TYPE "UDT_ConveyorStatistics"
TITLE = UDT_ConveyorStatistics
VERSION : 0.1
//User-defined structure of FB_Conveyor function block statistics.
   STRUCT
      EnergySave : "UDT_EventStatistic";   // Number of times that save energy mode occurs
      ConveyorUp : "UDT_EventStatistic";   // Conveyor up statistics
      ConveyorDown : "UDT_EventStatistic";   // Conveyor down statistics
      ConveyorStop : "UDT_EventStatistic";   // Conveyor down statistics
   END_STRUCT;

END_TYPE

TYPE "UDT_ConveyorStatus"
TITLE = UDT_ConveyorStatus
VERSION : 0.1
//User-defined structure of FB_Conveyor function block status.
   STRUCT
      Status : Int;   // Status number
      Specific : Struct
         Reverse { ExternalAccessible := 'False'; ExternalVisible := 'False'; ExternalWritable := 'False'} : Bool;   // Conveyor is running in reverse direction
      END_STRUCT;
   END_STRUCT;

END_TYPE

TYPE "UDT_EncoderStatisticsV2"
VERSION : 0.1
   STRUCT
      RunningFeedbackError : "UDT_EventStatistic";
      InvalidValue : "UDT_EventStatistic";
   END_STRUCT;

END_TYPE

TYPE "UDT_EncoderStatusV2"
VERSION : 0.1
   STRUCT
      InvalidValue : Bool;   // Invalid value
      RunningFeedbackError : Bool;   // Running feedback error
   END_STRUCT;

END_TYPE

TYPE "UDT_EncoderConfigurationV2"
VERSION : 0.1
   STRUCT
      EncoderMaxValue : DInt;   // The maximum value of the encoder where will rollover
      mmPerIncrement : Real;   // The mm per encoder incremental [mm]
      ErrorFilter : UDInt;   // Movment timeout without encoder data [ms]
      SamplingTime : UDInt;   // Save actual speed sampling time [ms]
   END_STRUCT;

END_TYPE

TYPE "UDT_EuchnerLockStatusV2"
VERSION : 0.1
   STRUCT
      LockFault : Bool;   // Internal lock fault
      DoorClosed : Bool;   // The door is closed
      DoorOpened : Bool;   // The door is opened
      BoltTongueClosed : Bool;   // The lock bolt tongue is closed
      ReqMissingAccessRights : Bool;   // Button access request triggered without permission from DHL
      ResetMissingAccessRights : Bool;   // Button reset triggered without permission from DHL
      DoorOpenedWithoutReq : Bool;   // Doors were opened without request and permission
      Safelylocked : Bool;   // The lock is safely locked
      SafetyLockAckReq : Bool;   // The safety lock signal needs to be confirmed
   END_STRUCT;

END_TYPE

TYPE "UDT_ConveyorCommand"
TITLE = UDT_ConveyorCommand
VERSION : 0.1
//User-defined structure of conveyor commands.
   STRUCT
      ManualMode { ExternalAccessible := 'False'; ExternalVisible := 'False'; ExternalWritable := 'False'} : Bool;   // Manual mode command from HMI
      ManualStartStop { ExternalAccessible := 'False'; ExternalVisible := 'False'; ExternalWritable := 'False'} : Bool;   // Run conveyor in manual mode
      ManualFullSpeed { ExternalAccessible := 'False'; ExternalVisible := 'False'; ExternalWritable := 'False'} : Bool;   // Full speed conveyor in manual mode
      ManualJog { ExternalAccessible := 'False'; ExternalVisible := 'False'; ExternalWritable := 'False'} : Bool;   // Command to jog conveyor in slow speed from HMI
      Reverse { ExternalAccessible := 'False'; ExternalVisible := 'False'; ExternalWritable := 'False'} : Bool;   // Command to run conveyor in reverse direction from HMI
      ManualSpeed : Int := 50;   // Manual mode speed as percentage of nominal speed [0-100%]
   END_STRUCT;

END_TYPE

TYPE "UDT_Outfeed2StatesConfiguration"
VERSION : 0.1
//User-defined structure of FB_Chute2PEC function block configuration.
   STRUCT
      FullDetectionTime : UDInt;   // Time after which chute full is detected
      FullReleaseTime : UDInt;   // Time after which chute full is released
      HalfFullDetectionTime : UDInt;   // Time after which chute half full is detected
      HalfFullReleaseTime : UDInt;   // Time after which chute half full is released
   END_STRUCT;

END_TYPE

TYPE "UDT_ConveyorConfiguration"
TITLE = UDT_ConveyorConfiguration
VERSION : 0.1
//User-defined structure of conveyor parameters.
   STRUCT
      Common : "UDT_ConveyorCommonConfiguration";   // Common configuration
      Forward_Direction : Struct   // Forward Direction configuration
         EnergySaveLenght : DInt;   // Distance conveyor travelled before energy save activate [cm]
         GapHeadToHead : DInt;   // Gapping head to head value [cm]
         GapTailToHead : DInt;   // Gapping tail to head value [cm]
         GapCorrection : DInt;   // Gap offset to cover VFD's ramps [cm]
         PEC_EoSDistanceOffset : DInt;   // Distance offset between photo eye and the end of conveyor [mm]
         Mode : Int;   // Automatic operation; 1- Slave; 2- Queue;
         FirstConveyorToStart { ExternalAccessible := 'False'; ExternalVisible := 'False'; ExternalWritable := 'False'} : Bool;   // First conveyor to start cascade mode forward direction
      END_STRUCT;
      Reverse_Direction : Struct   // Reverse Direction configuration
         EnergySaveLenght : DInt;   // Distance conveyor travelled before energy save activate [cm]
         GapHeadToHead : DInt;   // Gapping head to head value [cm]
         GapTailToHead : DInt;   // Gapping tail to head value [cm]
         GapCorrection : DInt;   // Gap offset to cover VFD's ramps [cm]
         PEC_BoSDistanceOffset : DInt;   // Distance offset between photo eye and the end of conveyor [mm]
         Mode : Int;   // Automatic operation; 1- Slave; 2- Queue;
         FirstConveyorToStart { ExternalAccessible := 'False'; ExternalVisible := 'False'; ExternalWritable := 'False'} : Bool;   // First conveyor to start cascade mode reverse direction
      END_STRUCT;
      CascadeTimeOnDelay : UDInt;   // Cascade time on delay [ms]
      ExtraGapRecovery : DInt;   // Extra gap to recovery die back [cm]
      SpeedSetpointLow : Int;   // Low speed setpoint [mm/s]
      SpeedSetpointNominal : Int;   // Nominal speed setpoint [mm/s]
      Energy { ExternalAccessible := 'False'; ExternalVisible := 'False'; ExternalWritable := 'False'} : Bool;   // Energy save mode enable
      Bi_Directional_Enable { ExternalAccessible := 'False'; ExternalVisible := 'False'; ExternalWritable := 'False'} : Bool;   // The conveyor can run in both directions
   END_STRUCT;

END_TYPE

TYPE "UDT_SerialCommunicationStatus"
VERSION : 0.1
   STRUCT
      ErrorCode : Word;   // Siemens Signal_Get error code - Check documetation
      Connected : Bool;   // Connected
      CommunicationFault : Bool;   // Communication fault
   END_STRUCT;

END_TYPE

TYPE "UDT_XrayInterface"
VERSION : 0.1
   STRUCT
      Backbelt : Struct   // Bacbelt function signals structure
         Enable : Bool;   // TRUE when Backbelt functionality for input conveyor is active
         Active : Bool;   // TRUE when Backbelt functionality activeted
      END_STRUCT;
      XrayConveyor : Struct   // Xray conveyor signals structure
         RunFwd : Bool;   // TRUE when conveyor is running forward
         RunRvs : Bool;   // TRUE when conveyor is running reverse
      END_STRUCT;
      InputConveyor : Struct   // Input conveyor signals structure
         CommandRunRvs : Bool;   // Request command to run reverse
      END_STRUCT;
      Communication : Struct   // SerialCommunication signals structure
         Connceted : Bool;   // Devices connected
         SendMessage : Struct   // Send message signal structure
            SendTrigger : Bool;   // Send message trigger
            GIN : Int;   // GIN number for new message
         END_STRUCT;
      END_STRUCT;
   END_STRUCT;

END_TYPE

FUNCTION_BLOCK "FB_VFD_MultiControl_V4"
{ S7_Optimized_Access := 'TRUE' }
AUTHOR : 'KBA-PM'
VERSION : 0.1
// ATTRIBUTES
// AUTO_NUMBER = True
// BLOCK_NUMBER = 107
// END_ATTRIBUTES
   VAR_INPUT
      i_UDT_VFDConfiguration { ExternalAccessible := 'False'; ExternalVisible := 'False'; ExternalWritable := 'False'} : "UDT_VFD_MultiControl_Configuration";   //   VFD configuration structure
      i_UDT_VFDInputs { ExternalAccessible := 'False'; ExternalVisible := 'False'; ExternalWritable := 'False'} : "UDT_VFD_MultiControl_PI";   //   VFD inputs structure
      ix_PowerOK { ExternalAccessible := 'False'; ExternalVisible := 'False'; ExternalWritable := 'False'} : Bool;   //   TRUE when External Power OK
      ix_SafetyOK { ExternalAccessible := 'False'; ExternalVisible := 'False'; ExternalWritable := 'False'} : Bool;   //   TRUE when Safety OK
      ix_SimulationModeActive { ExternalAccessible := 'False'; ExternalVisible := 'False'; ExternalWritable := 'False'} : Bool;   //   TRUE when Simulation mode active
   END_VAR

   VAR_OUTPUT
      q_UDT_HMIStatus { ExternalAccessible := 'False'; ExternalVisible := 'False'; ExternalWritable := 'False'} : "UDT_VfdStatus";   //   HMI status structure
      qsi_UDT_VFDSpeed { ExternalAccessible := 'False'; ExternalVisible := 'False'; ExternalWritable := 'False'} : SInt;   //   VFD speed setpoint
   END_VAR

   VAR_IN_OUT
      iq_UDT_ConveyorInterface : "UDT_ConveyorInterface";   //   Conveyor interface structure
      iq_UDT_VFDStatistics : "UDT_VfdStatistics";   //   Statistics structure
      iq_UDT_Equipment : "UDT_EquipmentControl";   //   Equipment structure
   END_VAR

   VAR
      s_FB_TimerOnOffDelayCheckSupply { ExternalAccessible := 'False'; ExternalVisible := 'False'; ExternalWritable := 'False'; S7_SetPoint := 'False'} : "FB_TimerOnOffDelay";   //  "TimerOnOffDelay" - to delay time for VFD supply contactor
      s_FB_TimerOnOffDelay_ProfinetNotOnlineMasking { ExternalAccessible := 'False'; ExternalVisible := 'False'; ExternalWritable := 'False'; S7_SetPoint := 'False'} : "FB_TimerOnOffDelay";   //   "TimerOnOffDelay" - to delay time for profinet not online masking
      s_FB_TimerOnOffDelay_ProfinetSlaveErrorMasking { ExternalAccessible := 'False'; ExternalVisible := 'False'; ExternalWritable := 'False'; S7_SetPoint := 'False'} : "FB_TimerOnOffDelay";   //   "TimerOnOffDelay" - to delay time for profinet error masking
      s_FB_TimerOnOffDelay_RunCommand_Motor_1 { ExternalAccessible := 'False'; ExternalVisible := 'False'; ExternalWritable := 'False'; S7_SetPoint := 'False'} : "FB_TimerOnOffDelay";   //   "TimerOnOffDelay" - to delay time for run command motor 1
      s_FB_TimerOnOffDelay_RunCommand_Motor_2 { ExternalAccessible := 'False'; ExternalVisible := 'False'; ExternalWritable := 'False'; S7_SetPoint := 'False'} : "FB_TimerOnOffDelay";   //   "TimerOnOffDelay" - to delay time for run command motor 2
      s_FB_TimerOnOffDelay_RunCommand_Motor_3 { ExternalAccessible := 'False'; ExternalVisible := 'False'; ExternalWritable := 'False'; S7_SetPoint := 'False'} : "FB_TimerOnOffDelay";   //   "TimerOnOffDelay" - to delay time for run command motor 3
      s_FB_TimerOnOffDelay_SafetyOK { ExternalAccessible := 'False'; ExternalVisible := 'False'; ExternalWritable := 'False'; S7_SetPoint := 'False'} : "FB_TimerOnOffDelay";   //   "TimerOnOffDelay" - to delay time for safety
      s_FB_TimerOnOffDelay_RunCommand_Motor_4 { ExternalAccessible := 'False'; ExternalVisible := 'False'; ExternalWritable := 'False'; S7_SetPoint := 'False'} : "FB_TimerOnOffDelay";   //   "TimerOnOffDelay" - to delay time for run command motor 4
      s_FB_TimerOnOffDelay_Instance { ExternalAccessible := 'False'; ExternalVisible := 'False'; ExternalWritable := 'False'; S7_SetPoint := 'False'} : "FB_TimerOnOffDelay";   //   "TimerOnOffDelay" - to delay time for Instance
      s_UDT_HMIStatus { ExternalAccessible := 'False'; ExternalVisible := 'False'; ExternalWritable := 'False'; S7_SetPoint := 'False'} : "UDT_VfdStatus";   //   HMI status structure
      s_UDT_PNDevice { ExternalAccessible := 'False'; ExternalVisible := 'False'; ExternalWritable := 'False'; S7_SetPoint := 'False'} : "UDT_PNDevice";   //   PN device info structure
      s_R_TRIG_RunForward {InstructionName := 'R_TRIG'; LibVersion := '1.0'; ExternalAccessible := 'False'; ExternalVisible := 'False'; ExternalWritable := 'False'; S7_SetPoint := 'False'} : R_TRIG;   //   Rising edge of Run forward signal
      s_R_TRIG_RunReverse {InstructionName := 'R_TRIG'; LibVersion := '1.0'; ExternalAccessible := 'False'; ExternalVisible := 'False'; ExternalWritable := 'False'; S7_SetPoint := 'False'} : R_TRIG;   //   Rising edge of Run reverse
      s_R_TRIG_PNSlaveNotOnline {InstructionName := 'R_TRIG'; LibVersion := '1.0'; ExternalAccessible := 'False'; ExternalVisible := 'False'; ExternalWritable := 'False'; S7_SetPoint := 'False'} : R_TRIG;   //   Rising edge for trigger Profinet slave not online statistics
      s_R_TRIG_PNSlaveError {InstructionName := 'R_TRIG'; LibVersion := '1.0'; ExternalAccessible := 'False'; ExternalVisible := 'False'; ExternalWritable := 'False'; S7_SetPoint := 'False'} : R_TRIG;   //   Rising edge for trigger Profinet slave error statistics
      s_R_TRIG_InternalError {InstructionName := 'R_TRIG'; LibVersion := '1.0'; ExternalAccessible := 'False'; ExternalVisible := 'False'; ExternalWritable := 'False'; S7_SetPoint := 'False'} : R_TRIG;   //   Rising edge for trigger Internal VFD Error statistics
      s_R_TRIG_Running {InstructionName := 'R_TRIG'; LibVersion := '1.0'; ExternalAccessible := 'False'; ExternalVisible := 'False'; ExternalWritable := 'False'; S7_SetPoint := 'False'} : R_TRIG;   //   Rising edge for starting of the running signal
      s_R_TRIG_Instance {InstructionName := 'R_TRIG'; LibVersion := '1.0'; ExternalAccessible := 'False'; ExternalVisible := 'False'; ExternalWritable := 'False'; S7_SetPoint := 'False'} : R_TRIG;   //   Raising edge for Instance
      s_R_TRIG_NewPNSlaveError {InstructionName := 'R_TRIG'; LibVersion := '1.0'; ExternalAccessible := 'False'; ExternalVisible := 'False'; ExternalWritable := 'False'; S7_SetPoint := 'False'} : R_TRIG;   //   New profinet slave error trigger
      s_R_TRIG_NewPNSlaveNotOnline {InstructionName := 'R_TRIG'; LibVersion := '1.0'; ExternalAccessible := 'False'; ExternalVisible := 'False'; ExternalWritable := 'False'; S7_SetPoint := 'False'} : R_TRIG;   //   New profinet slave not online trigger
      ss_RDREC { ExternalAccessible := 'False'; ExternalVisible := 'False'; ExternalWritable := 'False'} : Struct   //   Read error code record structure
         Valid { ExternalAccessible := 'False'; ExternalVisible := 'False'; ExternalWritable := 'False'} : Bool;   //      Read operation is done
         Busy { ExternalAccessible := 'False'; ExternalVisible := 'False'; ExternalWritable := 'False'} : Bool;   //      Read operation is in progress
         Error { ExternalAccessible := 'False'; ExternalVisible := 'False'; ExternalWritable := 'False'} : Bool;   //      Read operation has an error
         Status { ExternalAccessible := 'False'; ExternalVisible := 'False'; ExternalWritable := 'False'} : DWord;   //      Read operation status
         Lenght { ExternalAccessible := 'False'; ExternalVisible := 'False'; ExternalWritable := 'False'} : UInt;   //      Lenght of the read record
      END_STRUCT;
      ss_WRREC { ExternalAccessible := 'False'; ExternalVisible := 'False'; ExternalWritable := 'False'} : Struct   //   Write record structure
         Acceleration { ExternalAccessible := 'False'; ExternalVisible := 'False'; ExternalWritable := 'False'} : Struct   //      Acceleration
            REQ { ExternalAccessible := 'False'; ExternalVisible := 'False'; ExternalWritable := 'False'} : Bool;   //      Requirement
            Index { ExternalAccessible := 'False'; ExternalVisible := 'False'; ExternalWritable := 'False'} : DInt;   //      Index
            Done { ExternalAccessible := 'False'; ExternalVisible := 'False'; ExternalWritable := 'False'} : Bool;   //      Operation is done
            Busy { ExternalAccessible := 'False'; ExternalVisible := 'False'; ExternalWritable := 'False'} : Bool;   //      Write operation is in progress
            Error { ExternalAccessible := 'False'; ExternalVisible := 'False'; ExternalWritable := 'False'} : Bool;   //      Write operation has an error
            Status { ExternalAccessible := 'False'; ExternalVisible := 'False'; ExternalWritable := 'False'} : DWord;   //      Write operation status
            Data { ExternalAccessible := 'False'; ExternalVisible := 'False'; ExternalWritable := 'False'} : Word;   //      Data to write
         END_STRUCT;
         Deceleration { ExternalAccessible := 'False'; ExternalVisible := 'False'; ExternalWritable := 'False'} : Struct   //      Deceleration
            REQ { ExternalAccessible := 'False'; ExternalVisible := 'False'; ExternalWritable := 'False'} : Bool;   //      Requirement
            Index { ExternalAccessible := 'False'; ExternalVisible := 'False'; ExternalWritable := 'False'} : DInt;   //      Index
            Done { ExternalAccessible := 'False'; ExternalVisible := 'False'; ExternalWritable := 'False'} : Bool;   //      Operation is done
            Busy { ExternalAccessible := 'False'; ExternalVisible := 'False'; ExternalWritable := 'False'} : Bool;   //      Write operation is in progress
            Error { ExternalAccessible := 'False'; ExternalVisible := 'False'; ExternalWritable := 'False'} : Bool;   //      Write operation has an error
            Status { ExternalAccessible := 'False'; ExternalVisible := 'False'; ExternalWritable := 'False'} : DWord;   //      Write operation status
            Data { ExternalAccessible := 'False'; ExternalVisible := 'False'; ExternalWritable := 'False'} : Word;   //      Data to write
         END_STRUCT;
      END_STRUCT;
      ss_AccelerationDone { ExternalAccessible := 'False'; ExternalVisible := 'False'; ExternalWritable := 'False'} : Struct   //   Acceleration is written
         Motor_1 { ExternalAccessible := 'False'; ExternalVisible := 'False'; ExternalWritable := 'False'} : Bool;
         Motor_2 { ExternalAccessible := 'False'; ExternalVisible := 'False'; ExternalWritable := 'False'} : Bool;
         Motor_3 { ExternalAccessible := 'False'; ExternalVisible := 'False'; ExternalWritable := 'False'} : Bool;
         Motor_4 { ExternalAccessible := 'False'; ExternalVisible := 'False'; ExternalWritable := 'False'} : Bool;
         All { ExternalAccessible := 'False'; ExternalVisible := 'False'; ExternalWritable := 'False'} : Bool;
      END_STRUCT;
      ss_DecelerationDone { ExternalAccessible := 'False'; ExternalVisible := 'False'; ExternalWritable := 'False'} : Struct   //   Deceleration is written
         Motor_1 { ExternalAccessible := 'False'; ExternalVisible := 'False'; ExternalWritable := 'False'} : Bool;
         Motor_2 { ExternalAccessible := 'False'; ExternalVisible := 'False'; ExternalWritable := 'False'} : Bool;
         Motor_3 { ExternalAccessible := 'False'; ExternalVisible := 'False'; ExternalWritable := 'False'} : Bool;
         Motor_4 { ExternalAccessible := 'False'; ExternalVisible := 'False'; ExternalWritable := 'False'} : Bool;
         All { ExternalAccessible := 'False'; ExternalVisible := 'False'; ExternalWritable := 'False'} : Bool;
      END_STRUCT;
      s_VFDGeoStruct {InstructionName := 'GEOADDR'; LibVersion := '1.0'; ExternalAccessible := 'False'; ExternalVisible := 'False'; ExternalWritable := 'False'; S7_SetPoint := 'False'} : GEOADDR;   //   Geo structure indicate to telegram
      s_RDREC_ErrorCode {InstructionName := 'RDREC'; LibVersion := '1.0'; ExternalAccessible := 'False'; ExternalVisible := 'False'; ExternalWritable := 'False'; S7_SetPoint := 'False'} : RDREC;   //   Read error code record instruction
      s_WRREC_ACC {InstructionName := 'WRREC'; LibVersion := '1.1'; ExternalAccessible := 'False'; ExternalVisible := 'False'; ExternalWritable := 'False'; S7_SetPoint := 'False'} : WRREC;   //   Write acceleration record inctruction
      s_WRREC_DEC {InstructionName := 'WRREC'; LibVersion := '1.1'; ExternalAccessible := 'False'; ExternalVisible := 'False'; ExternalWritable := 'False'; S7_SetPoint := 'False'} : WRREC;   //   Write deceleration record instruction
      shw_VFD_Telegram { ExternalAccessible := 'False'; ExternalVisible := 'False'; ExternalWritable := 'False'} : HW_ANY;   //   Free telegram's HW_ID
      sr_MaximumSpeed { ExternalAccessible := 'False'; ExternalVisible := 'False'; ExternalWritable := 'False'} : Real;   //   Maximum speed [mm/s]
      sr_SpeedsetpointCorrected { ExternalAccessible := 'False'; ExternalVisible := 'False'; ExternalWritable := 'False'} : Real;   //   Speedsetpoint corrected with factor
      sw_ErrorCode { ExternalAccessible := 'False'; ExternalVisible := 'False'; ExternalWritable := 'False'} : Word;   //   VFD error code
      si_RequiredSpeedSetpoint { ExternalAccessible := 'False'; ExternalVisible := 'False'; ExternalWritable := 'False'} : Int;   //   Required speed setpoint
      si_ActualSpeed { ExternalAccessible := 'False'; ExternalVisible := 'False'; ExternalWritable := 'False'} : Int;   //   Actual speed in [mm/s]
      si_Log2GeoReturn { ExternalAccessible := 'False'; ExternalVisible := 'False'; ExternalWritable := 'False'} : Int;   //   Log2Geo function return
      si_Geo2LogReturn { ExternalAccessible := 'False'; ExternalVisible := 'False'; ExternalWritable := 'False'} : Int;   //   Geo2Log function return
      si_AccelerationSetpoint { ExternalAccessible := 'False'; ExternalVisible := 'False'; ExternalWritable := 'False'} : Int;   //   Acceleration setpoint value
      si_DecelerationSetpoint { ExternalAccessible := 'False'; ExternalVisible := 'False'; ExternalWritable := 'False'} : Int;   //   Deceleration setpoint value
      si_AccelerationOld { ExternalAccessible := 'False'; ExternalVisible := 'False'; ExternalWritable := 'False'} : Int;   //   Old acceleration value
      si_DecelerationOld { ExternalAccessible := 'False'; ExternalVisible := 'False'; ExternalWritable := 'False'} : Int;   //   Old deceleration value
      si_MotorNumber_Acc { ExternalAccessible := 'False'; ExternalVisible := 'False'; ExternalWritable := 'False'} : Int;   //   Motor number that is connected to the Multicontrol module [1,2,3 or 4]
      si_MotorNumber_Dec { ExternalAccessible := 'False'; ExternalVisible := 'False'; ExternalWritable := 'False'} : Int;   //   Motor number that is connected to the Multicontrol module [1,2,3 or 4]
      si_PNSlaveErrorCount { ExternalAccessible := 'False'; ExternalVisible := 'False'; ExternalWritable := 'False'} : Int;   //   Profinet slave error counter
      si_PNSlaveNotOnlineCount { ExternalAccessible := 'False'; ExternalVisible := 'False'; ExternalWritable := 'False'} : Int;   //   Profinet slave not online counter
      ssi_MotorSpeed { ExternalAccessible := 'False'; ExternalVisible := 'False'; ExternalWritable := 'False'} : SInt;   //   Motor speed value
      sx_ConfigurationError { ExternalAccessible := 'False'; ExternalVisible := 'False'; ExternalWritable := 'False'} : Bool;   //   Commissioning: configuration error
      sx_PNDeviceHealthy { ExternalAccessible := 'False'; ExternalVisible := 'False'; ExternalWritable := 'False'} : Bool;   //   Profinet device is online and error free
      sx_PowerOk { ExternalAccessible := 'False'; ExternalVisible := 'False'; ExternalWritable := 'False'} : Bool;   //   Communication, safety and power are available
      sx_VFD_Available { ExternalAccessible := 'False'; ExternalVisible := 'False'; ExternalWritable := 'False'} : Bool;   //   Hardware of VFD is ok
      sx_ErrorActive { ExternalAccessible := 'False'; ExternalVisible := 'False'; ExternalWritable := 'False'} : Bool;   //   Block has an error
      sx_MotorError { ExternalAccessible := 'False'; ExternalVisible := 'False'; ExternalWritable := 'False'} : Bool;   //   Motor error all
      sx_Motor_1_Error { ExternalAccessible := 'False'; ExternalVisible := 'False'; ExternalWritable := 'False'} : Bool;   //   Motor error 1
      sx_Motor_2_Error { ExternalAccessible := 'False'; ExternalVisible := 'False'; ExternalWritable := 'False'} : Bool;   //   Motor error 2
      sx_Motor_3_Error { ExternalAccessible := 'False'; ExternalVisible := 'False'; ExternalWritable := 'False'} : Bool;   //   Motor error 3
      sx_Motor_4_Error { ExternalAccessible := 'False'; ExternalVisible := 'False'; ExternalWritable := 'False'} : Bool;   //   Motor error 4
      sx_EnableOperation { ExternalAccessible := 'False'; ExternalVisible := 'False'; ExternalWritable := 'False'} : Bool;   //   Enable operation signal
      sx_RunVFDForward { ExternalAccessible := 'False'; ExternalVisible := 'False'; ExternalWritable := 'False'} : Bool;   //   Start VFD forward
      sx_RunVFDReverse { ExternalAccessible := 'False'; ExternalVisible := 'False'; ExternalWritable := 'False'} : Bool;   //   Start VFD backward
      sx_SpeedSetpointReached { ExternalAccessible := 'False'; ExternalVisible := 'False'; ExternalWritable := 'False'} : Bool;   //   Motor is running at requested speed
      sx_ErrorDone { ExternalAccessible := 'False'; ExternalVisible := 'False'; ExternalWritable := 'False'} : Bool;   //   Error code is read
      sx_SafetyOK { ExternalAccessible := 'False'; ExternalVisible := 'False'; ExternalWritable := 'False'} : Bool;   //   Safety ok
      sx_MaskingReset { ExternalAccessible := 'False'; ExternalVisible := 'False'; ExternalWritable := 'False'} : Bool;   //   Masking reset
      sx_PNSlaveError { ExternalAccessible := 'False'; ExternalVisible := 'False'; ExternalWritable := 'False'} : Bool;   //   Profinet slave error
      sx_PNSlaveNotOnline { ExternalAccessible := 'False'; ExternalVisible := 'False'; ExternalWritable := 'False'} : Bool;   //   Profinet slave not online
   END_VAR

   VAR CONSTANT
      ci_VFDArea : UInt := 1;   //   Area ID of IO Profinet devices
      ci_SubmoduleHWType : UInt := 5;   //   Submodule HW_type number
      ci_TelegramSlot : UInt := 2;   //   Free Siemens telegram slot
      ci_TelegramSubslot : UInt := 1;   //   Free Siemens telegram subslot
      cdi_ErrorCodeIndex : DInt := 17154;   //   Error code index
      cdi_AccelerationIndex : DInt := 18200;   //   Acceleration index
      cdi_DecelerationIndex : DInt := 18204;   //   Deceleration index
   END_VAR


BEGIN
	(*
	----------------------------------------------------------------------------------------
	|                                                                                      |
	|  Copyright  2023             FORTNA Europe BV                                        |
	|  All Rights Reserved         Netherlands                                             |
	|                                                                                      |
	----------------------------------------------------------------------------------------

	Version history:
	Date        | Version   | Author        | Remark
	----------------------------------------------------------------------------------------
	24/05/2023  | 1.0       | S.Nikodem     | Initial version for 4 motors | DHL Munich 2023
	13/03/2024  | 1.1       | S. Nieswiec   | Added to new baseline
	*)

	REGION 1 - Get Device Profinet number

	    // Getting information about Profinet Device.
	    "FC_GetDevicePN"(is_PNDeviceName := #i_UDT_VFDConfiguration.VFDPNDeviceName,
	                     ix_SimulationModeActive := #ix_SimulationModeActive,
	                     iqUDT_PND := #s_UDT_PNDevice);

	END_REGION

	REGION 2 - Motor validation

	    //Motor number 1
	    // Delay
	    #s_FB_TimerOnOffDelay_RunCommand_Motor_1(iudi_OnDelayTime := 1500,
	                                             ix_SignalToDelay :=
	                                             (#sx_RunVFDForward
	                                             OR #sx_RunVFDReverse)
	                                             AND #i_UDT_VFDInputs.CurrentMotor1 < #i_UDT_VFDConfiguration.MinimumCurrentWhenRunninng);

	    #ssi_MotorSpeed := #i_UDT_VFDInputs.SpeedMotor1;

	    IF (#s_FB_TimerOnOffDelay_RunCommand_Motor_1.qx_DelayedSignal AND #sx_EnableOperation) OR #i_UDT_VFDInputs.ErrorMotor1
	    THEN

	        #sx_Motor_1_Error := TRUE;

	    END_IF;

	    //Motor number 2
	    #s_FB_TimerOnOffDelay_RunCommand_Motor_2(iudi_OnDelayTime := 1500,
	                                             ix_SignalToDelay :=
	                                             (#sx_RunVFDForward
	                                             OR #sx_RunVFDReverse)
	                                             AND #i_UDT_VFDInputs.CurrentMotor2 < #i_UDT_VFDConfiguration.MinimumCurrentWhenRunninng);

	    #ssi_MotorSpeed := #i_UDT_VFDInputs.SpeedMotor2;

	    IF (#s_FB_TimerOnOffDelay_RunCommand_Motor_2.qx_DelayedSignal AND #sx_EnableOperation) OR #i_UDT_VFDInputs.ErrorMotor2

	    THEN

	        #sx_Motor_2_Error := TRUE;

	    END_IF;

	    //Motor number 3
	    #s_FB_TimerOnOffDelay_RunCommand_Motor_3(iudi_OnDelayTime := 1500,
	                                             ix_SignalToDelay :=
	                                             (#sx_RunVFDForward
	                                             OR #sx_RunVFDReverse)
	                                             AND #i_UDT_VFDInputs.CurrentMotor3 < #i_UDT_VFDConfiguration.MinimumCurrentWhenRunninng);

	    #ssi_MotorSpeed := #i_UDT_VFDInputs.SpeedMotor3;

	    IF (#s_FB_TimerOnOffDelay_RunCommand_Motor_3.qx_DelayedSignal AND #sx_EnableOperation) OR #i_UDT_VFDInputs.ErrorMotor3
	    THEN

	        #sx_Motor_3_Error := TRUE;

	    END_IF;

	    //Motor number 4
	    #s_FB_TimerOnOffDelay_RunCommand_Motor_4(iudi_OnDelayTime := 1500,
	                                             ix_SignalToDelay :=
	                                             (#sx_RunVFDForward
	                                             OR #sx_RunVFDReverse)
	                                             AND #i_UDT_VFDInputs.CurrentMotor4 < #i_UDT_VFDConfiguration.MinimumCurrentWhenRunninng);

	    #ssi_MotorSpeed := #i_UDT_VFDInputs.SpeedMotor4;

	    IF (#s_FB_TimerOnOffDelay_RunCommand_Motor_4.qx_DelayedSignal AND #sx_EnableOperation) OR #i_UDT_VFDInputs.ErrorMotor4
	    THEN

	        #sx_Motor_4_Error := TRUE;

	    END_IF;

	    //Collect errors from all motors
	    #sx_MotorError := #sx_Motor_1_Error OR #sx_Motor_2_Error OR #sx_Motor_3_Error OR #sx_Motor_4_Error;

	END_REGION

	REGION 3 - Reset errors

	    // Reset the errors on the command from the conveyor interface.
	    //
	    #s_R_TRIG_Instance(CLK := #ix_SafetyOK,
	                       Q => #sx_SafetyOK);

	    #s_FB_TimerOnOffDelay_Instance(iudi_OffDelayTime := 10000,
	                                   ix_SignalToDelay := #sx_SafetyOK,
	                                   qx_DelayedSignal => #sx_MaskingReset);


	    IF #iq_UDT_ConveyorInterface.InternalErrorReset
	        OR (#sx_MaskingReset
	        AND "DB_Memory".Clock_2Hz)
	    THEN
	        #s_UDT_HMIStatus.PNSlaveNotonline := FALSE;
	        #s_UDT_HMIStatus.PNSlaveError := FALSE;
	        #s_UDT_HMIStatus.InternalError := FALSE;
	        #sx_MotorError := FALSE;
	        #sx_Motor_1_Error := FALSE;
	        #sx_Motor_2_Error := FALSE;
	        #sx_Motor_3_Error := FALSE;
	        #sx_Motor_4_Error := FALSE;

	    END_IF;

	END_REGION

	REGION 4 - Hardware check

	    //Auto reset for Profinet errors, when inactive the masking time is 0
	    IF NOT #i_UDT_VFDConfiguration.AutoReset THEN

	        #i_UDT_VFDConfiguration.TimePNErrorMasking := 0;

	    END_IF;

	    // Hardware will be available only after the delay, so the device has time for the initialization.
	    #s_FB_TimerOnOffDelayCheckSupply(iudi_OnDelayTime := 2000,
	                                     ix_SignalToDelay := #ix_PowerOK,
	                                     qx_DelayedSignal => #sx_PowerOk);

	    #s_FB_TimerOnOffDelay_ProfinetNotOnlineMasking(iudi_OnDelayTime := #i_UDT_VFDConfiguration.TimePNErrorMasking,
	                                                   iudi_OffDelayTime := 0,
	                                                   ix_SignalToDelay := #sx_PNSlaveNotOnline,
	                                                   qx_DelayedSignal => #s_UDT_HMIStatus.PNSlaveNotonline);

	    #s_FB_TimerOnOffDelay_ProfinetSlaveErrorMasking(iudi_OnDelayTime := #i_UDT_VFDConfiguration.TimePNErrorMasking,
	                                                    iudi_OffDelayTime := 0,
	                                                    ix_SignalToDelay := #sx_PNSlaveError,
	                                                    qx_DelayedSignal => #s_UDT_HMIStatus.PNSlaveError);

	    #s_R_TRIG_NewPNSlaveNotOnline(CLK := #sx_PNSlaveNotOnline);
	    #s_R_TRIG_NewPNSlaveError(CLK := #sx_PNSlaveError);
	    // Check if PN device is online.
	    IF NOT "DB_ProfinetDiagnostic".ProfinetNetworks[#s_UDT_PNDevice.PNNetworknumber].DeviceStatus[#s_UDT_PNDevice.PNDeviceNumber].DeviceState.Exist
	        AND NOT #ix_SimulationModeActive
	        AND #sx_PowerOk
	    THEN
	        #sx_PNSlaveNotOnline := TRUE;
	        #iq_UDT_Equipment.Command.Reset := "DB_Memory".Clock_1Hz AND #i_UDT_VFDConfiguration.AutoReset;
	    ELSE
	        #sx_PNSlaveNotOnline := FALSE;
	    END_IF;

	    IF #s_R_TRIG_NewPNSlaveNotOnline.Q THEN
	        #si_PNSlaveNotOnlineCount += 1;
	    END_IF;

	    // Check if PN device has an error.
	    IF "DB_ProfinetDiagnostic".ProfinetNetworks[#s_UDT_PNDevice.PNNetworknumber].DeviceStatus[#s_UDT_PNDevice.PNDeviceNumber].DeviceState.Error
	        AND NOT #ix_SimulationModeActive
	        AND #sx_PowerOk
	    THEN
	        #sx_PNSlaveError := TRUE;
	        #iq_UDT_Equipment.Command.Reset := "DB_Memory".Clock_1Hz AND #i_UDT_VFDConfiguration.AutoReset;
	    ELSE
	        #sx_PNSlaveError := FALSE;
	    END_IF;

	    IF #s_R_TRIG_NewPNSlaveError.Q THEN
	        #si_PNSlaveErrorCount += 1;
	    END_IF;

	    // Set bit when PN device is healthy (online and no error).
	    #sx_PNDeviceHealthy :=
	    NOT #s_UDT_HMIStatus.PNSlaveNotonline
	    AND NOT #s_UDT_HMIStatus.PNSlaveError
	    AND #s_UDT_PNDevice.PNDeviceFound
	    AND #sx_PowerOk;

	    // Set VFD available bit when all conditions are met.
	    #sx_VFD_Available :=
	    (NOT #sx_MotorError
	    AND #sx_PowerOk
	    AND #sx_PNDeviceHealthy)
	    OR #ix_SimulationModeActive;

	END_REGION

	REGION 5 - Extract telegram's HW_ID

	    // Extract telegram's HW_ID
	    #si_Log2GeoReturn := LOG2GEO(LADDR := "DB_ProfinetDiagnostic".ProfinetNetworks[#s_UDT_PNDevice.PNNetworknumber].DeviceStatus[#s_UDT_PNDevice.PNDeviceNumber].DeviceState.HW_ID, GEOADDR := #s_VFDGeoStruct);
	    #s_VFDGeoStruct.AREA := #ci_VFDArea;
	    #s_VFDGeoStruct.HWTYPE := #ci_SubmoduleHWType;
	    #s_VFDGeoStruct.STATION := INT_TO_UINT(#s_UDT_PNDevice.PNDeviceNumber);
	    #s_VFDGeoStruct.SLOT := #ci_TelegramSlot;
	    #s_VFDGeoStruct.SUBSLOT := #ci_TelegramSubslot;

	    #si_Geo2LogReturn := GEO2LOG(GEOADDR := #s_VFDGeoStruct, LADDR => #shw_VFD_Telegram);

	END_REGION

	REGION 6 - Check errors

	    #s_FB_TimerOnOffDelay_SafetyOK(iudi_OnDelayTime := 10000,
	                                   ix_SignalToDelay := #ix_SafetyOK);

	    // Check if the motor has an error.
	    IF #s_FB_TimerOnOffDelay_SafetyOK.qx_DelayedSignal  //#ix_SafetyOK
	    THEN
	        #s_UDT_HMIStatus.InternalError := #sx_MotorError;

	    END_IF;
	    // Create trigger on error.
	    #s_R_TRIG_InternalError(CLK := #s_UDT_HMIStatus.InternalError);

	    // If the internal error occured, reset the error code read done signal.
	    IF #s_R_TRIG_InternalError.Q
	    THEN
	        #sx_ErrorDone := FALSE;
	    END_IF;

	    // If there is an internal error, read the error code from the Interroll VFD. Otherwise, reset it.
	    IF NOT #s_UDT_HMIStatus.InternalError
	    THEN
	        #s_UDT_HMIStatus.ErrorCode := 0;
	    ELSE
	        // Read the error code from the multicontrol.
	        #s_RDREC_ErrorCode(REQ := ((NOT #sx_ErrorDone OR "mx_FirstScan") AND NOT #s_UDT_HMIStatus.PNSlaveNotonline),
	                           ID := #shw_VFD_Telegram,
	                           INDEX := #cdi_ErrorCodeIndex,
	                           MLEN := 0,
	                           VALID => #ss_RDREC.Valid,
	                           BUSY => #ss_RDREC.Busy,
	                           ERROR => #ss_RDREC.Error,
	                           STATUS => #ss_RDREC.Status,
	                           LEN => #ss_RDREC.Lenght,
	                           RECORD := #sw_ErrorCode);

	        // IF error code is read, set the error code read signal and write it to the structure.
	        IF #s_RDREC_ErrorCode.VALID
	        THEN
	            #sx_ErrorDone := TRUE;
	            #s_UDT_HMIStatus.ErrorCode := WORD_TO_INT(SWAP_WORD(IN := #sw_ErrorCode));
	        END_IF;
	    END_IF;

	END_REGION

	REGION 7 - Check if configuration is ok for commissioning purposes

	    // Validate the VFD configuration and motor number.
	    IF #i_UDT_VFDConfiguration.MaximumSpeed > 0.0
	    THEN
	        #sx_ConfigurationError := FALSE;
	    ELSE
	        #sx_ConfigurationError := TRUE;
	    END_IF;

	END_REGION

	REGION 8 - Handle speed

	    // Write max speed to static.
	    #sr_MaximumSpeed := #i_UDT_VFDConfiguration.MaximumSpeed;

	    // Use correction factor to calculate setpint for diaginal use
	    #sr_SpeedsetpointCorrected := INT_TO_REAL(#iq_UDT_ConveyorInterface.SpeedSetpoint) * #i_UDT_VFDConfiguration.CorrectionFactor;

	    // Actual speed setpoint
	    #si_RequiredSpeedSetpoint := REAL_TO_INT((#sr_SpeedsetpointCorrected * 100.0) / (#sr_MaximumSpeed));

	    // Speed setpoint saturation in case when the speed setpoint is higher than the max speed.
	    IF #si_RequiredSpeedSetpoint > 100
	    THEN
	        #si_RequiredSpeedSetpoint := 100;
	        #iq_UDT_ConveyorInterface.ConfigurationError := TRUE;
	    ELSIF #si_RequiredSpeedSetpoint < -100
	    THEN
	        #si_RequiredSpeedSetpoint := -100;
	        #iq_UDT_ConveyorInterface.ConfigurationError := TRUE;
	    END_IF;

	END_REGION

	REGION 9 - Prepare output data VFD

	    REGION 9.1 - Set speed setpoint in forward and reverse direction
	        // Get rising edge of Run forward and reverse signal.
	        #s_R_TRIG_RunForward(CLK := #iq_UDT_ConveyorInterface.RunFwd);
	        #s_R_TRIG_RunReverse(CLK := #iq_UDT_ConveyorInterface.RunRvs);

	        // When rising edge of the forward or reverse signal is received, the drive has to stop to be able to make the switch.
	        IF #s_R_TRIG_RunForward.Q
	            OR #s_R_TRIG_RunReverse.Q
	        THEN
	            #qsi_UDT_VFDSpeed := 0;
	        END_IF;

	        // If motor stopped and Run forward is requested and forward direction is interlock, set run forward signal and reset run reverse signal.
	        IF //#ssi_MotorSpeed = 0 and
	            #iq_UDT_ConveyorInterface.RunFwd
	            AND #i_UDT_VFDConfiguration.InterlockFwd
	        THEN
	            #sx_RunVFDForward := TRUE;
	            #sx_RunVFDReverse := FALSE;
	        END_IF;

	        // If motor stopped and Run reverse is requested and reverse direction is interlock, set run reverse signal and reset run forward signal.
	        IF // #ssi_MotorSpeed = 0 AND
	            #iq_UDT_ConveyorInterface.RunRvs
	            AND #i_UDT_VFDConfiguration.InterlockRvs
	        THEN
	            #sx_RunVFDReverse := TRUE;
	            #sx_RunVFDForward := FALSE;
	        END_IF;

	    END_REGION

	    REGION 9.2 - Stopping

	        // Stop the VFD if one of the following conditions is met.
	        IF (NOT #iq_UDT_ConveyorInterface.RunRvs AND NOT #iq_UDT_ConveyorInterface.RunFwd)
	            OR (#iq_UDT_ConveyorInterface.RunRvs AND #iq_UDT_ConveyorInterface.RunFwd)
	            OR (#sx_RunVFDReverse AND NOT #i_UDT_VFDConfiguration.InterlockRvs)
	            OR (#sx_RunVFDForward AND NOT #i_UDT_VFDConfiguration.InterlockFwd)
	            OR ((#s_R_TRIG_RunForward.Q AND #ssi_MotorSpeed < 0)
	            OR (#s_R_TRIG_RunReverse.Q AND #ssi_MotorSpeed > 0))
	        THEN
	            #sx_RunVFDReverse := FALSE;
	            #sx_RunVFDForward := FALSE;
	        END_IF;

	    END_REGION

	    REGION 9.3 - Check for enable operation signal

	        // Operation is enable when VFD is available and there is one of the run commands.
	        #sx_EnableOperation :=
	        #sx_VFD_Available
	        AND (#sx_RunVFDForward OR #sx_RunVFDReverse)
	        AND NOT #sx_ConfigurationError;

	    END_REGION

	END_REGION

	REGION 10 - Write outputs to VFD

	    REGION 10.1 - Write speed setpoint to drive

	        // The conveyor stopped and may now run in forward direction.
	        IF ((#sx_RunVFDForward AND NOT #i_UDT_VFDConfiguration.DirectionReversal)
	            OR (#sx_RunVFDReverse AND #i_UDT_VFDConfiguration.DirectionReversal))
	            AND #sx_EnableOperation
	        THEN
	            #qsi_UDT_VFDSpeed := INT_TO_SINT(#si_RequiredSpeedSetpoint);
	        END_IF;

	        // The conveyor stopped and may now run in reverse direction.
	        IF ((#sx_RunVFDReverse AND NOT #i_UDT_VFDConfiguration.DirectionReversal)
	            OR (#sx_RunVFDForward AND #i_UDT_VFDConfiguration.DirectionReversal))
	            AND #sx_EnableOperation
	        THEN
	            #qsi_UDT_VFDSpeed := - INT_TO_SINT(#si_RequiredSpeedSetpoint);
	        END_IF;

	        // Clear speed setpoint when run isn't request.
	        IF (NOT #sx_RunVFDForward
	            AND NOT #sx_RunVFDReverse)
	            OR NOT #sx_EnableOperation
	        THEN
	            #qsi_UDT_VFDSpeed := 0;
	        END_IF;

	    END_REGION


	    REGION 10.2 - Calculate acceleration and deceleration values

	        // Recalculating Acceleration ramp - deviding maximum configured speed by Ramp up time and devide it by 1000.
	        #si_AccelerationSetpoint := REAL_TO_INT(#sr_MaximumSpeed / (UDINT_TO_REAL(#i_UDT_VFDConfiguration.VFDRampUpTime) / 1000.0));

	        // Recalculating Deceleration ramp - deviding maximum configured speed by Ramp down time and devide it by 1000.
	        #si_DecelerationSetpoint := REAL_TO_INT(#sr_MaximumSpeed / (UDINT_TO_REAL(#i_UDT_VFDConfiguration.VFDRampDownTime) / 1000.0));

	    END_REGION

	    REGION 10.3 - Write acceleration to drive


	        REGION 10.3.1 - Acceleration write operation is done.

	            IF #ss_AccelerationDone.All
	            THEN
	                // There is new acceleration value or device is offline.
	                IF #si_AccelerationSetpoint <> #si_AccelerationOld
	                    OR NOT #s_UDT_HMIStatus.PNSlaveNotonline
	                THEN
	                    // Reset the accleration operation done signal.
	                    #ss_AccelerationDone.Motor_1 := FALSE;
	                    #ss_AccelerationDone.Motor_2 := FALSE;
	                    #ss_AccelerationDone.Motor_3 := FALSE;
	                    #ss_AccelerationDone.Motor_4 := FALSE;
	                    #ss_AccelerationDone.All := FALSE;
	                END_IF;
	            END_IF;

	        END_REGION


	        // The acceleration operation isn't done or there is first scan and device is online.
	        IF (NOT #ss_AccelerationDone.All OR "mx_FirstScan")
	            AND NOT #s_UDT_HMIStatus.PNSlaveNotonline
	        THEN

	            //Set motor number
	            IF NOT #ss_AccelerationDone.Motor_1 THEN
	                #si_MotorNumber_Acc := 1;
	            ELSIF NOT #ss_AccelerationDone.Motor_2 THEN
	                #si_MotorNumber_Acc := 2;
	            ELSIF NOT #ss_AccelerationDone.Motor_3 THEN
	                #si_MotorNumber_Acc := 3;
	            ELSIF NOT #ss_AccelerationDone.Motor_4 THEN
	                #si_MotorNumber_Acc := 4;
	            ELSE
	                #si_MotorNumber_Acc := 0;
	            END_IF;

	            // There isn't an  acceleration equal to 0.
	            IF #si_AccelerationSetpoint > 0 THEN

	                // Calculate the index of the acceleration.
	                #ss_WRREC.Acceleration.Index := #cdi_AccelerationIndex + #si_MotorNumber_Acc;
	                // Prepare the data.
	                #ss_WRREC.Acceleration.Data := SWAP(INT_TO_WORD(#si_AccelerationSetpoint));
	                // Set operation is required.
	                #ss_WRREC.Acceleration.REQ := TRUE;

	                // Send acceleration to the device.
	                #s_WRREC_ACC(REQ := #ss_WRREC.Acceleration.REQ,
	                             ID := #shw_VFD_Telegram,
	                             INDEX := #ss_WRREC.Acceleration.Index,
	                             LEN := 0,
	                             DONE => #ss_WRREC.Acceleration.Done,
	                             BUSY => #ss_WRREC.Acceleration.Busy,
	                             ERROR => #ss_WRREC.Acceleration.Error,
	                             STATUS => #ss_WRREC.Acceleration.Status,
	                             RECORD := #ss_WRREC.Acceleration.Data);

	                // Send operation is done.
	                IF #ss_WRREC.Acceleration.Done
	                THEN
	                    // Reset operation is required bit.
	                    #ss_WRREC.Acceleration.REQ := FALSE;

	                    // Set the operation is done signal.
	                    CASE #si_MotorNumber_Acc OF
	                        1:
	                            #ss_AccelerationDone.Motor_1 := TRUE;

	                        2:
	                            #ss_AccelerationDone.Motor_1 := TRUE;

	                        3:
	                            #ss_AccelerationDone.Motor_1 := TRUE;

	                        4:
	                            #ss_AccelerationDone.Motor_1 := TRUE;
	                            #ss_AccelerationDone.All := TRUE;
	                    END_CASE;

	                    // Write acceleration value into the old one.
	                    #si_AccelerationOld := #si_AccelerationSetpoint;
	                END_IF;
	            END_IF;
	        END_IF;

	    END_REGION

	    REGION 10.4 - Write deceleration to drive

	        // Deceleration write operation is done.
	        IF #ss_DecelerationDone.All
	        THEN
	            // There is new deceleration value or device is offline.
	            IF #si_DecelerationSetpoint <> #si_DecelerationOld
	                OR NOT #s_UDT_HMIStatus.PNSlaveNotonline
	            THEN
	                // Reset the deceleration operation done signal.
	                #ss_DecelerationDone.Motor_1 := FALSE;
	                #ss_DecelerationDone.Motor_2 := FALSE;
	                #ss_DecelerationDone.Motor_3 := FALSE;
	                #ss_DecelerationDone.Motor_4 := FALSE;
	                #ss_DecelerationDone.All := FALSE;

	            END_IF;
	        END_IF;

	        // The deceleration operation isn't done or there is first scan and device is online.
	        IF NOT #ss_DecelerationDone.All OR "mx_FirstScan"
	            AND NOT #s_UDT_HMIStatus.PNSlaveNotonline
	        THEN
	            // There isn't an  deceleration equal to 0.
	            IF #si_DecelerationSetpoint > 0 THEN

	                //Set motor number
	                IF NOT #ss_DecelerationDone.Motor_1 THEN
	                    #si_MotorNumber_Dec := 1;
	                ELSIF NOT #ss_DecelerationDone.Motor_2 THEN
	                    #si_MotorNumber_Dec := 2;
	                ELSIF NOT #ss_DecelerationDone.Motor_3 THEN
	                    #si_MotorNumber_Dec := 3;
	                ELSIF NOT #ss_DecelerationDone.Motor_4 THEN
	                    #si_MotorNumber_Dec := 4;
	                ELSE
	                    #si_MotorNumber_Dec := 0;
	                END_IF;

	                // Calculate the index of the deceleration.
	                #ss_WRREC.Deceleration.Index := #cdi_DecelerationIndex + #si_MotorNumber_Dec;
	                // Prepare the data.
	                #ss_WRREC.Deceleration.Data := SWAP(INT_TO_WORD(#si_DecelerationSetpoint));
	                // Set operation is required.
	                #ss_WRREC.Deceleration.REQ := TRUE;

	                // Send deceleration to the device.
	                #s_WRREC_DEC(REQ := #ss_WRREC.Deceleration.REQ,
	                             ID := #shw_VFD_Telegram,
	                             INDEX := #ss_WRREC.Deceleration.Index,
	                             LEN := 0,
	                             DONE => #ss_WRREC.Deceleration.Done,
	                             BUSY => #ss_WRREC.Deceleration.Busy,
	                             ERROR => #ss_WRREC.Deceleration.Error,
	                             STATUS => #ss_WRREC.Deceleration.Status,
	                             RECORD := #ss_WRREC.Deceleration.Data);

	                // Send operation is done.
	                IF #ss_WRREC.Deceleration.Done
	                THEN
	                    // Reset operation is required bit.
	                    #ss_WRREC.Deceleration.REQ := FALSE;

	                    // Set the operation is done signal.
	                    CASE #si_MotorNumber_Dec OF
	                        1:
	                            #ss_DecelerationDone.Motor_1 := TRUE;

	                        2:
	                            #ss_DecelerationDone.Motor_1 := TRUE;

	                        3:
	                            #ss_DecelerationDone.Motor_1 := TRUE;

	                        4:
	                            #ss_DecelerationDone.Motor_1 := TRUE;
	                            #ss_DecelerationDone.All := TRUE;
	                    END_CASE;

	                    // Write deceleration value into the old one.
	                    #si_DecelerationOld := #si_DecelerationSetpoint;
	                END_IF;
	            END_IF;
	        END_IF;

	    END_REGION

	END_REGION

	REGION 11 - Copy signals to interface DB and to status output UDT

	    // Create collective error.
	    #sx_ErrorActive :=
	    #s_UDT_HMIStatus.PNSlaveNotonline
	    OR #s_UDT_HMIStatus.PNSlaveError
	    OR #s_UDT_HMIStatus.InternalError
	    OR #sx_ConfigurationError;

	    // Motor is giving direct signal on start, move setpoint to actual speed.
	    IF #ssi_MotorSpeed <> 0
	    THEN
	        #si_ActualSpeed := #iq_UDT_ConveyorInterface.SpeedSetpoint;
	        #sx_SpeedSetpointReached := TRUE;
	    ELSE
	        #si_ActualSpeed := 0;
	        #sx_SpeedSetpointReached := FALSE;
	    END_IF;

	    // Write interface bits.
	    #iq_UDT_ConveyorInterface.VFDRunning :=
	    #sx_VFD_Available
	    AND #iq_UDT_ConveyorInterface.ActualSpeed <> 0;

	    // Speed setpoint is reached.
	    #iq_UDT_ConveyorInterface.VFDatSpeed :=
	    #sx_SpeedSetpointReached
	    AND #sx_VFD_Available;

	    // Set the internal VFD error bit if any fault is active.
	    #iq_UDT_ConveyorInterface.InternalErrorVFD := #sx_ErrorActive;
	    // Copy the speed value to the output.
	    #iq_UDT_ConveyorInterface.ActualSpeed := #si_ActualSpeed;

	    // Copy error status to output.
	    #q_UDT_HMIStatus := #s_UDT_HMIStatus;

	END_REGION

	REGION 12 - Statistics

	    // Create trigger on error and create statistics for profinet slave not online.
	    #s_R_TRIG_PNSlaveNotOnline(CLK := #s_UDT_HMIStatus.PNSlaveNotonline);

	    IF #iq_UDT_ConveyorInterface.ResetStatistics
	        OR #s_UDT_HMIStatus.PNSlaveNotonline
	    THEN
	        "FC_Statistics"(ix_Reset := #iq_UDT_ConveyorInterface.ResetStatistics,
	                        ix_Activate := #s_UDT_HMIStatus.PNSlaveNotonline,
	                        ix_RTrigActivate := #s_R_TRIG_PNSlaveNotOnline.Q,
	                        iqUDT_Statistics := #iq_UDT_VFDStatistics.PNSlaveNotOnline);
	    END_IF;

	    // Create trigger on error and create statistics for profinet slave error.
	    #s_R_TRIG_PNSlaveError(CLK := #s_UDT_HMIStatus.PNSlaveError);

	    IF #iq_UDT_ConveyorInterface.ResetStatistics
	        OR #s_UDT_HMIStatus.PNSlaveError
	    THEN
	        "FC_Statistics"(ix_Reset := #iq_UDT_ConveyorInterface.ResetStatistics,
	                        ix_Activate := #s_UDT_HMIStatus.PNSlaveError,
	                        ix_RTrigActivate := #s_R_TRIG_PNSlaveError.Q,
	                        iqUDT_Statistics := #iq_UDT_VFDStatistics.PNSlaveError);
	    END_IF;

	    IF #iq_UDT_ConveyorInterface.ResetStatistics
	        OR #s_UDT_HMIStatus.InternalError
	    THEN
	        "FC_Statistics"(ix_Reset := #iq_UDT_ConveyorInterface.ResetStatistics,
	                        ix_Activate := #s_UDT_HMIStatus.InternalError,
	                        ix_RTrigActivate := #s_R_TRIG_InternalError.Q,
	                        iqUDT_Statistics := #iq_UDT_VFDStatistics.VFDInternalError);
	    END_IF;

	    // Create trigger on running signal and create statistics for running status.
	    #s_R_TRIG_Running(CLK := #iq_UDT_ConveyorInterface.VFDRunning);

	    IF #iq_UDT_ConveyorInterface.ResetStatistics
	        OR #iq_UDT_ConveyorInterface.VFDRunning
	    THEN
	        "FC_Statistics"(ix_Reset := #iq_UDT_ConveyorInterface.ResetStatistics,
	                        ix_Activate := #iq_UDT_ConveyorInterface.VFDRunning,
	                        ix_RTrigActivate := #s_R_TRIG_Running.Q,
	                        iqUDT_Statistics := #iq_UDT_VFDStatistics.Running);
	    END_IF;

	END_REGION
END_FUNCTION_BLOCK

TYPE "UDT_ConveyorHandshake"
TITLE = UDT_ConveyorHandshake
VERSION : 0.1
//User-defined structure of conveyor handshake variables.
   STRUCT
      GIN : Int;   // General identification number
      NrOfPosToShift : Int;   // Number of positions to shift
      DownstreamDisplacement : Int;   // Displacement from downstream [cm]
      RTS { ExternalAccessible := 'False'; ExternalVisible := 'False'; ExternalWritable := 'False'} : Bool;   // Conveyor ready to send
      RTR { ExternalAccessible := 'False'; ExternalVisible := 'False'; ExternalWritable := 'False'} : Bool;   // Conveyor ready to receive
      TIP { ExternalAccessible := 'False'; ExternalVisible := 'False'; ExternalWritable := 'False'} : Bool;   // Transfer in progress
      ResetEnergySave { ExternalAccessible := 'False'; ExternalVisible := 'False'; ExternalWritable := 'False'} : Bool;   // Reset energy save mode
      CascadeStartUp { ExternalAccessible := 'False'; ExternalVisible := 'False'; ExternalWritable := 'False'} : Bool;   // Cascade startup
      ReqStop { ExternalAccessible := 'False'; ExternalVisible := 'False'; ExternalWritable := 'False'} : Bool;   // Request stop
   END_STRUCT;

END_TYPE

TYPE "UDT_OutfeedStatus"
VERSION : 0.1
   STRUCT
      ID : UInt := 0;   // ID
      NotAvailable : Bool;   // Collect signal - TRUE when outfeed not available
      Full : Bool;   // Outfeed full , impossible to send next parcels.
      Disable : Bool;   // Deactivated by the operator from the HMI or MFC
   END_STRUCT;

END_TYPE

TYPE "UDT_ArmDiverterConfiguration"
VERSION : 0.1
   STRUCT
      VerticalConveyorMode : Int;   // [1]Continuous operation if the main conveyor is running; [2]Operation if arm is not in Home position.
      ArmDiverterSpeedSetpointLow : Int;   // Arm diverter low speed setpoint [mm/s]
      ArmDiverterSpeedSetpointNominal : Int;   // Arm diverter nominal speed setpoint [mm/s]
      DischargeLocationID : UInt;   // Discharge Location ID
      OutfeedsNumber : UInt;   // OutfeedsNumber [1 ..5]
      DecisionPoint : Int;   // Decision Point - Distance from the end of the conveyor [cm]
      DecisionParcelWindow : Int;   // Decision window - Maximum distance from the beginning of the parcel to the "Decision point"
      AssociatedConveyorLength : DInt;   // Associated conveyor length
      ParcelFreeWindow : Int;   // Distance from the end of the parcel that must be left empty to sort the parcel correctly
      ParcelFreeWindowStart : Int;   // Start point in tracking data -  Window in which the package must not be in order to start the arm [cm]
      ParcelFreeWindowEnd : Int;   // End point in tracking data - Window in which the package must not be in order to start the arm [cm]
      DataTransferPoint : Int;   // Transfer point to the exit conveyor [cm]
      MaximumMovementTime : UDInt;   // Maximum time to move [ms]
      JogNoHornTime : UDInt;   // Time within jog buttons can be pressed without new startup indication [ms]
      MaximumParcelDivertTime : UDInt;   // Maximum parcel divert time [ms]
      Sensor : Struct   // Sensors on/off time configuration
         PRX_HomeTimeOnDelay { ExternalAccessible := 'False'; ExternalVisible := 'False'; ExternalWritable := 'False'} : UDInt;   // Proxy sensor home position on delay [ms]
         PRX_HomeTimeOffDelay : UDInt;   // Proxy sensor home position off delay [ms]
         PRX_DivertTimeOnDelay { ExternalAccessible := 'False'; ExternalVisible := 'False'; ExternalWritable := 'False'} : UDInt;   // Proxy sensor divert position on delay [ms]
         PRX_DivertTimeOffDelay : UDInt;   // Proxy sensor divert position off delay [ms]
         LS_HomeTimeOnDelay : UDInt;   // Limit switch home position on delay [ms]
         LS_HomeTimeOffDelay : UDInt;   // Limit switch home position off delay [ms]
         LS_DivertTimeOnDelay : UDInt;   // Limit switch divert position on delay [ms]
         LS_DivertTimeOffDelay : UDInt;   // Limit switch divert position off delay [ms]
         PRX_BRK_HomeTimeOnDelay : UDInt;   // Brake sensor home position on delay [ms]
         PRX_BRK_HomeTimeOffDelay : UDInt;   // Brake sensor home position off delay [ms]
         PRX_BRK_DivertTimeOnDelay : UDInt;   // Brake sensor divert position on delay [ms]
         PRX_BRK_DivertTimeOffDelay : UDInt;   // Brake sensor divert position off delay [ms]
      END_STRUCT;
   END_STRUCT;

END_TYPE

TYPE "UDT_ArmDiverterCommand"
VERSION : 0.1
   STRUCT
      ManualMode : Bool;   // Manual mode command from HMI
      ManualHomePosition : Bool;   // Manual mode command go to home position
      ManualDivertPosition : Bool;   // Manual mode command go to divert position
      JogHomePosition : Bool;   // Jog command go to home position
      JogDivertPosition : Bool;   // Jog command go to divert position
      Reset : Bool;   // Reset command
   END_STRUCT;

END_TYPE

FUNCTION_BLOCK "FB_ConnectionCheck"
{ S7_Optimized_Access := 'TRUE' }
VERSION : 3.2
// ATTRIBUTES
// AUTO_NUMBER = True
// BLOCK_NUMBER = 205
// END_ATTRIBUTES
   VAR_INPUT
      ib_Watchdog { ExternalAccessible := 'False'; ExternalVisible := 'False'; ExternalWritable := 'False'} : Byte;   // Input watchdog
      ix_Trigger100ms { ExternalAccessible := 'False'; ExternalVisible := 'False'; ExternalWritable := 'False'} : Bool;   // Cycled 100 ms trigger
   END_VAR

   VAR_OUTPUT
      qb_Watchdog { ExternalAccessible := 'False'; ExternalVisible := 'False'; ExternalWritable := 'False'} : Byte;   // Generated watchdog
   END_VAR

   VAR_IN_OUT
      iqudt_ConnectionStatus : "UDT_ConnectStatus";   // Connection status
   END_VAR

   VAR
      s_FB_ConnectionFaultTimerOnDelay { ExternalAccessible := 'False'; ExternalVisible := 'False'; ExternalWritable := 'False'; S7_SetPoint := 'False'} : "FB_TimerOnOffDelay";   // Connection fault timer on delay
      sb_InWatchdogOld { ExternalAccessible := 'False'; ExternalVisible := 'False'; ExternalWritable := 'False'} : Byte;   // Watch dog old
      sb_GeneratedWatchdog { ExternalAccessible := 'False'; ExternalVisible := 'False'; ExternalWritable := 'False'} : Byte;   // Generated watchdog
      sx_SetConnectionFaultTimer { ExternalAccessible := 'False'; ExternalVisible := 'False'; ExternalWritable := 'False'} : Bool;   // Set connection fault timer
      sx_ConnectionFault { ExternalAccessible := 'False'; ExternalVisible := 'False'; ExternalWritable := 'False'} : Bool;   // Connection faulr
   END_VAR

   VAR CONSTANT
      cudi_ConnectionFaultOnDelay : UDInt := 10000;   // Connection On Delay
   END_VAR


BEGIN
	(*
	----------------------------------------------------------------------------------------
	|                                                                                      |
	|  Copyright  2023             FORTNA Europe BV                                        |
	|  All Rights Reserved         Netherlands                                             |
	|                                                                                      |
	----------------------------------------------------------------------------------------

	Version history:
	Date        | Version   | Author        | Remark
	----------------------------------------------------------------------------------------
	31/03/2022  | 3.0       | M. Piela      | First release TIA 16
	06/09/2023  | 3.1       | S. Nikodem    | Added watchdog generations on output
	11/09/2023  | 3.2       | S. Theocharis | Corrected variable prefixes
	*)

	REGION 1 - Connection check

	    #sx_SetConnectionFaultTimer := (#ib_Watchdog = #sb_InWatchdogOld);

	    IF #ib_Watchdog <> #sb_InWatchdogOld
	    THEN
	        #sb_InWatchdogOld := #ib_Watchdog;
	    END_IF;

	    #s_FB_ConnectionFaultTimerOnDelay(iudi_OnDelayTime := #cudi_ConnectionFaultOnDelay,
	                                      ix_SignalToDelay := #sx_SetConnectionFaultTimer,
	                                      ix_Enable := TRUE,
	                                      qx_DelayedSignal => #sx_ConnectionFault);

	END_REGION

	REGION 2 - Status update

	    #iqudt_ConnectionStatus.Specific.CommunicationFault := #sx_ConnectionFault;
	    #iqudt_ConnectionStatus.Specific.Connected := NOT #sx_ConnectionFault;

	    IF #sx_ConnectionFault
	    THEN
	        #iqudt_ConnectionStatus.Status := "DB_HMIStatusConfiguration".CommunicationError;
	    END_IF;

	    IF NOT #sx_ConnectionFault
	    THEN
	        #iqudt_ConnectionStatus.Status := "DB_HMIStatusConfiguration".AutoON;
	    END_IF;

	END_REGION

	REGION 3 - Watchdog generations

	    //Watchdog counter to be updated after every 100 msec
	    IF #ix_Trigger100ms THEN

	        IF #sb_GeneratedWatchdog >= 255 OR #sb_GeneratedWatchdog < 0
	        THEN
	            #sb_GeneratedWatchdog := 0;
	        END_IF;

	        #sb_GeneratedWatchdog := INT_TO_BYTE(BYTE_TO_INT(#sb_GeneratedWatchdog) + 1);

	    END_IF;

	    //Copy value
	    #qb_Watchdog := #sb_GeneratedWatchdog;

	END_REGION
END_FUNCTION_BLOCK

FUNCTION_BLOCK "FB_MFC_Sort_COY_RegInfo"
{ S7_Optimized_Access := 'TRUE' }
VERSION : 0.1
// ATTRIBUTES
// AUTO_NUMBER = True
// BLOCK_NUMBER = 116
// END_ATTRIBUTES
   VAR_INPUT
      is_ObjectID : String[10];   // Parcel identifier
      ii_XrayLocation : Int;   // X-ray location
      ii_SourceNode : Int;   // ID Source Node
      ii_DestinationNode : Int;   // ID Destination Node
   END_VAR

   VAR_OUTPUT
      qx_Error : Bool;   // TRUE when collective block error occurred
      qx_Warning : Bool;   // TRUE when collective block warning occurred
   END_VAR

   VAR_IN_OUT
      iq_UDT_FifoHeader : "UDT_FifoHeader";   // FIFO header
      iqa_FifoData : Array[*] of "UDT_MessageV2";   // FIFO data buffer
      iqi_MessageSequenceNumber : Int;   // Message number
   END_VAR

   VAR
      ss_FB_HeartbeatPulse : "FB_Pulse";   // Heartbeat send pulse generator
      s_UDT_MessageArray : "UDT_MessageV2";   // Message array byte
      s_UDT_MessageHeader : "UDT_MFCSortMessageHeader";   // Message header
      ss_MessageBody : Struct   // Message body
         MsgID : Word;   // Message ID
         MsgLength : Word;   // Message length
         ObjectID : DWord;   // Parcel identifier
         XrayLocation : Word;
         Eom : Byte;   // End of message
      END_STRUCT;
      ss_Status : Struct   // Status structure
         FIFOStatus : "UDT_FifoStatus";
         FIFOError { S7_SetPoint := 'True'} : Bool;   //  FIFO error
         FIFOWarning { S7_SetPoint := 'True'} : Bool;   // FIFO warning
         InvalidMessageArraySize : Bool;   // Message array is too short for message
         InvalidTimeInterval : Bool;   // Heartbeat time interval lower than zero
      END_STRUCT;
      si_Old_Object_ID : String[10];   // Value from previous PLC cycle
      sdi_SerializePosition : DInt;   // Position in array where serialize finished writing data +1
      si_MaximumMessageLength : Int;   // Maximum number of elements in message array
      si_SerializeStatus : Int;   // Function serialize status
      sx_NewData : Bool;   // True - send a message to the MFC
   END_VAR

   VAR_TEMP
      tudi_Temp : UDInt;   // temporarry variable
   END_VAR

   VAR CONSTANT
      ci_MessageLength : Word := 16#0008;   // 10#0008 = 16#0008 - Message length
      ci_MsgID : Word := 16#0136;   // 10#0310 = 16#0136 - Message ID
      ci_MsgLength : Word := 16#0004;   // 10#0004 = 16#0004 - Message length
      ci_Som : Byte := 16#FD;   // Start of message
      ci_Eom : Byte := 16#FE;   // End of message
   END_VAR


BEGIN
	(*
	----------------------------------------------------------------------------------------
	|                                                                                      |
	|  Copyright  2023             FORTNA Europe BV                                        |
	|  All Rights Reserved         Netherlands                                             |
	|                                                                                      |
	----------------------------------------------------------------------------------------
	Version history:
	Date        | Version   | Author       | Remark
	----------------------------------------------------------------------------------------
	24/05/2023  | 1.0       | S. Nikodem   | Release TIA 17 | DHL Munich 2023
	13/03/2023  | 1.1       | S. Nieswiec  | Updated for new Baseline
	*)

	REGION 1 – FIFO header status update

	    // Mode 'S' - FIFO register status update.
	    "FC_Fifo"(ic_Mode := 'S',
	              qUDT_Status => #ss_Status.FIFOStatus,
	              qx_Error => #ss_Status.FIFOError,
	              qx_Warning => #ss_Status.FIFOWarning,
	              iqv_Data := #s_UDT_MessageArray,
	              iqUDT_FifoHeader := #iq_UDT_FifoHeader,
	              iqv_DataBuffer := #iqa_FifoData);

	END_REGION

	REGION 2 – Data preparation

	    //Send message when is new parcel
	    #sx_NewData := (#is_ObjectID <> #si_Old_Object_ID) AND NOT (#is_ObjectID = '');
	    // Save last value
	    #si_Old_Object_ID := #is_ObjectID;

	END_REGION

	REGION 3 – Message array size validation

	    // Get size of the array.
	    #si_MaximumMessageLength := "FC_GetNrOfArrayEl"(#s_UDT_MessageArray.Bytes);

	    // Message array size validation.
	    #ss_Status.InvalidMessageArraySize := WORD_TO_INT(#ci_MessageLength) > #si_MaximumMessageLength;

	END_REGION


	REGION 4 – Message preparation

	    // FIFO full check.
	    IF NOT #iq_UDT_FifoHeader.Status.Full
	    THEN
	        // Errors and send pulse check.
	        IF NOT #ss_Status.FIFOError
	            AND NOT #ss_Status.InvalidMessageArraySize
	            AND #sx_NewData
	        THEN

	            REGION 4.1 – Header preparation

	                // Check sequence number. If it is equal or greater than 255 reset it to 1.
	                IF #iqi_MessageSequenceNumber <= 255
	                THEN
	                    #iqi_MessageSequenceNumber += 1;
	                ELSE
	                    #iqi_MessageSequenceNumber := 1;
	                END_IF;

	                // Write parts of the header into structure.
	                #s_UDT_MessageHeader.SOM := #ci_Som;
	                #s_UDT_MessageHeader.SourceNode := INT_TO_BYTE(#ii_SourceNode);
	                #s_UDT_MessageHeader.DestinationNode := INT_TO_BYTE(#ii_DestinationNode);
	                #s_UDT_MessageHeader.SeqNumber := INT_TO_BYTE(#iqi_MessageSequenceNumber);
	                #s_UDT_MessageHeader.DataLength := #ci_MessageLength;
	                #s_UDT_MessageHeader.NumMsg := 1;

	                //Convert string value to UDINT
	                #tudi_Temp := STRING_TO_UDINT(#is_ObjectID);

	                // Write parts of the body into structure.
	                #ss_MessageBody.MsgID := #ci_MsgID;
	                #ss_MessageBody.MsgLength := #ci_MsgLength;
	                #ss_MessageBody.ObjectID := UDINT_TO_DWORD(#tudi_Temp);
	                #ss_MessageBody.XrayLocation := INT_TO_WORD(#ii_XrayLocation);
	                #ss_MessageBody.Eom := #ci_Eom;

	            END_REGION

	            REGION 4.2 – Convert message into array of bytes

	                // Initialize the header serialize position and convert header structure into array of bytes.
	                #sdi_SerializePosition := 0;
	                #si_SerializeStatus := Serialize(SRC_VARIABLE := #s_UDT_MessageHeader,
	                                                 DEST_ARRAY => #s_UDT_MessageArray.Bytes,
	                                                 POS := #sdi_SerializePosition);

	                // Initialize the body serialize position and convert header structure into array of bytes
	                #si_SerializeStatus := Serialize(SRC_VARIABLE := #ss_MessageBody,
	                                                 DEST_ARRAY => #s_UDT_MessageArray.Bytes,
	                                                 POS := #sdi_SerializePosition);

	            END_REGION

	            REGION 4.3 – Write message into the FIFO buffer

	                // Mode 'W' - Write FIFO record.
	                "FC_Fifo"(ic_Mode := 'W',
	                          qUDT_Status => #ss_Status.FIFOStatus,
	                          qx_Error => #ss_Status.FIFOError,
	                          qx_Warning => #ss_Status.FIFOWarning,
	                          iqv_Data := #s_UDT_MessageArray,
	                          iqUDT_FifoHeader := #iq_UDT_FifoHeader,
	                          iqv_DataBuffer := #iqa_FifoData);

	            END_REGION

	        END_IF;
	    ELSE
	        // If FIFO is full set FIFO main and FIFO full errors.
	        #ss_Status.FIFOError := TRUE;
	        #ss_Status.FIFOStatus.FifoFull := TRUE;
	    END_IF;

	END_REGION

	REGION 5 - Status

	    // Parametrization collective error output.
	    #qx_Error :=
	    #ss_Status.FIFOError
	    OR #ss_Status.InvalidTimeInterval
	    OR #ss_Status.InvalidMessageArraySize;

	    // Parametrization collective warning output.
	    #qx_Warning := #ss_Status.FIFOWarning;

	END_REGION
END_FUNCTION_BLOCK

TYPE "UDT_DownStream_Sorter_Common"
VERSION : 0.1
   STRUCT
      Watchdog { ExternalAccessible := 'False'; ExternalVisible := 'False'; ExternalWritable := 'False'} : Byte;
      FireAlarm : Bool;
   END_STRUCT;

END_TYPE

TYPE "UDT_Sorter_DownStream_Common"
VERSION : 0.1
   STRUCT
      Watchdog { ExternalAccessible := 'False'; ExternalVisible := 'False'; ExternalWritable := 'False'} : Byte;
      AvailableCarriers { ExternalAccessible := 'False'; ExternalVisible := 'False'; ExternalWritable := 'False'} : Int;
      SignalManagement { ExternalAccessible := 'False'; ExternalVisible := 'False'; ExternalWritable := 'False'} : Bool;
   END_STRUCT;

END_TYPE

FUNCTION_BLOCK "FB_MFC_Sort_SortResult"
{ S7_Optimized_Access := 'TRUE' }
VERSION : 0.1
// ATTRIBUTES
// AUTO_NUMBER = True
// BLOCK_NUMBER = 124
// END_ATTRIBUTES
   VAR_INPUT
      is_ObjectID : String[10];   // Parcel identifier
      ii_DischargeLocation : UInt;   // Discharge location identifier
      ii_Result : Int;   // 1 = Sorted, 2 = Rejected, 3 = Lost
      ii_Reason : Int;   // 0 = Unknown, 1 = Success, 2 = Chute full, 3 = Chute not available, 4 = Unload failed, 5 = Late destination, 6 = Item lost, 7 = Higher priority available
      ii_SourceNode { ExternalAccessible := 'False'; ExternalVisible := 'False'; ExternalWritable := 'False'} : Int := 0;   // Source Node
      ii_DestinationNode { ExternalAccessible := 'False'; ExternalVisible := 'False'; ExternalWritable := 'False'} : Int := 0;   // Destination Node
   END_VAR

   VAR_OUTPUT
      qx_Error : Bool;   // TRUE when collective block error occurred
      qx_Warning : Bool;   // TRUE when collective block warning occurred
   END_VAR

   VAR_IN_OUT
      iq_UDT_FifoHeader : "UDT_FifoHeader";   // FIFO header
      iqs_FifoData : Array[*] of "UDT_MessageV2";   // FIFO data buffer
      iqdi_MessageSequenceNumber : Int;   // Message number
   END_VAR

   VAR
      s_UDT_MessageArray : "UDT_MessageV2";   // Message array byte
      s_UDT_MessageHeader : "UDT_MFCSortMessageHeader";   // Message header
      ss_MessageBody : Struct   // Message body
         MsgID : Word;   // Message ID
         MsgLength : Word;   // Message length
         Object_ID : String[10];   // Parcel identifier
         DischargeLocation : Word;   // Discharge location identifier
         Result : Byte;   // 0 = Sorted, 1 = Rejected, 2 = Lost
         Reason : Byte;   // 0 = Success, 1 = Chute full, 2 = Chute not available, 3 = Unload failed, 4 = Late destination, 5 = Item lost, 6 = Unknown
         Eom : Byte;   // End of message
      END_STRUCT;
      ss_Status : Struct   // Status structure
         FIFOStatus : "UDT_FifoStatus";
         FIFOError { S7_SetPoint := 'True'} : Bool;   //  FIFO error
         FIFOWarning { S7_SetPoint := 'True'} : Bool;   // FIFO warning
         InvalidMessageArraySize : Bool;   // Message array is too short for message
         InvalidTimeInterval : Bool;   // Heartbeat time interval lower than zero
      END_STRUCT;
      sdi_SerializePosition : DInt;   // Position in array where serialize finished writing data +1
      si_MaximumMessageLength : Int;   // Maximum number of elements in message array
      si_SerializeStatus : Int;   // Function serialize status
   END_VAR

   VAR CONSTANT
      ci_MessageLength : Word := 16#000C;   // 10#0012 = 16#000C - Message length
      ci_Som : Byte := 16#FD;   // Start of message
      ci_Eom : Byte := 16#FE;   // End of message
      ci_MsgID : Word := 16#00CB;   // 10#0203 = 16#00CB - Message ID
      ci_MsgLength : Word := 16#0008;   // 10#0008 = 16#0008 - Message length
   END_VAR


BEGIN
	(*
	----------------------------------------------------------------------------------------
	|                                                                                      |
	|  Copyright  2023             FORTNA Europe BV                                        |
	|  All Rights Reserved         Netherlands                                             |
	|                                                                                      |
	----------------------------------------------------------------------------------------
	Version history:
	Date        | Version   | Author       | Remark
	----------------------------------------------------------------------------------------
	29/06/2023  | 1.0       | S. Nikodem   | Release TIA 17 | DHL Munich 2023
	13/03/2023  | 1.1       | S. Nieswiec  | Updated for new Baseline
	02/05/2024  | 1.2       | J.Majer      | Datatype conversions changed from automatic to explicit, to accomodate IEC 61131-3 standard

	*)

	REGION 1 – FIFO header status update

	    // Mode 'S' - FIFO register status update.
	    "FC_Fifo"(ic_Mode := 'S',
	              qUDT_Status => #ss_Status.FIFOStatus,
	              qx_Error => #ss_Status.FIFOError,
	              qx_Warning => #ss_Status.FIFOWarning,
	              iqv_Data := #s_UDT_MessageArray,
	              iqUDT_FifoHeader := #iq_UDT_FifoHeader,
	              iqv_DataBuffer := #iqs_FifoData);

	END_REGION

	REGION 2 – Data preparation

	END_REGION

	REGION 3 – Message array size validation

	    // Get size of the array.
	    #si_MaximumMessageLength := "FC_GetNrOfArrayEl"(#s_UDT_MessageArray.Bytes);

	    // Message array size validation.
	    #ss_Status.InvalidMessageArraySize := WORD_TO_INT(#ci_MessageLength) > #si_MaximumMessageLength;

	END_REGION

	REGION 4 – Message preparation

	    // FIFO full check.
	    IF NOT #iq_UDT_FifoHeader.Status.Full
	    THEN
	        // Errors and send pulse check.
	        IF NOT #ss_Status.FIFOError
	            AND NOT #ss_Status.InvalidMessageArraySize
	        THEN

	            REGION 4.1 – Header preparation

	                // Check sequence number. If it is equal or greater than 255 reset it to 1.
	                IF #iqdi_MessageSequenceNumber <= 255
	                THEN
	                    #iqdi_MessageSequenceNumber += 1;
	                ELSE
	                    #iqdi_MessageSequenceNumber := 1;
	                END_IF;

	                // Write parts of the header into structure.
	                #s_UDT_MessageHeader.SOM := #ci_Som;
	                #s_UDT_MessageHeader.SourceNode := INT_TO_BYTE(#ii_SourceNode);
	                #s_UDT_MessageHeader.DestinationNode := INT_TO_BYTE(#ii_DestinationNode);
	                #s_UDT_MessageHeader.SeqNumber := INT_TO_BYTE(#iqdi_MessageSequenceNumber);
	                #s_UDT_MessageHeader.DataLength := #ci_MessageLength;
	                #s_UDT_MessageHeader.NumMsg := 1;

	                // Write parts of the body into structure.
	                #ss_MessageBody.MsgID := #ci_MsgID;
	                #ss_MessageBody.MsgLength := #ci_MsgLength;
	                #ss_MessageBody.Object_ID := #is_ObjectID;
	                #ss_MessageBody.DischargeLocation := UINT_TO_WORD(#ii_DischargeLocation);
	                #ss_MessageBody.Result := INT_TO_BYTE(#ii_Result);
	                #ss_MessageBody.Reason := INT_TO_BYTE(#ii_Reason);
	                #ss_MessageBody.Eom := #ci_Eom;

	            END_REGION

	            REGION 4.2 – Convert message into array of bytes

	                // Initialize the header serialize position and convert header structure into array of bytes.
	                #sdi_SerializePosition := 0;
	                #si_SerializeStatus := Serialize(SRC_VARIABLE := #s_UDT_MessageHeader,
	                                                 DEST_ARRAY => #s_UDT_MessageArray.Bytes,
	                                                 POS := #sdi_SerializePosition);

	                // Initialize the body serialize position and convert header structure into array of bytes
	                #si_SerializeStatus := Serialize(SRC_VARIABLE := #ss_MessageBody,
	                                                 DEST_ARRAY => #s_UDT_MessageArray.Bytes,
	                                                 POS := #sdi_SerializePosition);

	            END_REGION

	            REGION 4.3 – Write message into the FIFO buffer

	                // Mode 'W' - Write FIFO record.
	                "FC_Fifo"(ic_Mode := 'W',
	                          qUDT_Status => #ss_Status.FIFOStatus,
	                          qx_Error => #ss_Status.FIFOError,
	                          qx_Warning => #ss_Status.FIFOWarning,
	                          iqv_Data := #s_UDT_MessageArray,
	                          iqUDT_FifoHeader := #iq_UDT_FifoHeader,
	                          iqv_DataBuffer := #iqs_FifoData);

	            END_REGION

	        END_IF;
	    ELSE
	        // If FIFO is full set FIFO main and FIFO full errors.
	        #ss_Status.FIFOError := TRUE;
	        #ss_Status.FIFOStatus.FifoFull := TRUE;
	    END_IF;

	END_REGION

	REGION 5 - Status

	    // Parametrization collective error output.
	    #qx_Error :=
	    #ss_Status.FIFOError
	    OR #ss_Status.InvalidTimeInterval
	    OR #ss_Status.InvalidMessageArraySize;

	    // Parametrization collective warning output.
	    #qx_Warning := #ss_Status.FIFOWarning;

	END_REGION
END_FUNCTION_BLOCK

TYPE "UDT_SerialCommunicationSendStatus"
VERSION : 0.1
   STRUCT
      Done : Bool;   // Status from Send_P2P function
      Error : Bool;   // Status from Send_P2P function
      Status : Word;   // Status from Send_P2P function
      WrongMessageLength : Bool;   // Wrong prepared message length
   END_STRUCT;

END_TYPE

TYPE "UDT_ArmDiverterStatus"
VERSION : 0.1
   STRUCT
      Status : Int;   // Status number
      Specific : Struct   // Equipment specific warnings and errors
         TimeoutError : Bool;   // Arm movement timed out
         LimitHomeError : Bool;   // Limit swich sensor error
         LimitDivertError : Bool;   // Limit swich sensor error
         PXHomeError : Bool;   // Proxy sensor error
         PXDivertError : Bool;   // Proxy sensor error
         AtHomePosition : Bool;   // Arm is in home position
         AtDivertPosition : Bool;   // Arm is in divert position
         ReferencError : Bool;   // Referencing error - the arm is not detected by any sensor.
         ParcelDivertError : Bool;   // Parcel diversion error, time too long
         JamExitSensor : Bool;   // Jam on Exit sensor
      END_STRUCT;
   END_STRUCT;

END_TYPE

FUNCTION_BLOCK "FB_MFC_Sort_VIDResponse_ASCII"
{ S7_Optimized_Access := 'TRUE' }
VERSION : 0.1
// ATTRIBUTES
// AUTO_NUMBER = True
// BLOCK_NUMBER = 129
// END_ATTRIBUTES
   VAR_INPUT
      is_ObjectID : String[10];   // Parcel identifier
      ii_SorterID : Int;   // Sorter identifier
      i_ActualTimeDTL {InstructionName := 'DTL'; LibVersion := '1.0'} : DTL;   // Actual date and time in DTL
   END_VAR

   VAR_OUTPUT
      qx_Error : Bool;   // TRUE when collective block error occurred
      qx_Warning : Bool;   // TRUE when collective block warning occurred
   END_VAR

   VAR_IN_OUT
      iq_UDT_FifoHeader : "UDT_FifoHeader";   // FIFO header
      iqs_FifoData : Array[*] of "UDT_MessageV2";   // FIFO data buffer
      iqdi_MessageSequenceNumber : Int;   // Message number
   END_VAR

   VAR
      s_UDT_MessageArray : "UDT_MessageV2";   // Message array byte
      s_UDT_MessageHeader : "UDT_MFCSortMessageHeader";   // Message header
      ss_MessageBody : Struct   // Message body
         MsgID : Word;   // Message ID
         MsgLength : Word;   // Message length
         ObjectID : String[10];   // Parcel identifier
         VID : Array[0..15] of Byte;   // Virtual Item Identifier
         Eom : Byte;   // End of message
      END_STRUCT;
      ss_Status : Struct   // Status structure
         FIFOStatus : "UDT_FifoStatus";
         HTAReturn : Struct   // Status structure from HTA function
            Month : Word;   // HTA_Month
            Day : Word;   // HTA_Day
         END_STRUCT;
         FIFOError { S7_SetPoint := 'True'} : Bool;   //  FIFO error
         FIFOWarning { S7_SetPoint := 'True'} : Bool;   // FIFO warning
         InvalidMessageArraySize : Bool;   // Message array is too short for message
         InvalidTimeInterval : Bool;   // Heartbeat time interval lower than zero
         InvalidInputData : Bool;   // Input is not in range
      END_STRUCT;
      ss_VID : String;   // Virtual Item Identifier
      sa_VIDBytes : Array[1..16] of Byte;   // VID  - array with data in ASCII
      sdi_SerializePosition : DInt;   // Position in array where serialize finished writing data +1
      sdi_VIDCode : DInt;   // VID Code
      si_MaximumMessageLength : Int;   // Maximum number of elements in message array
      si_SerializeStatus : Int;   // Function serialize status
      ss_OldObjectID : String[10];   // Value from previous PLC cycle
      sx_NewData : Bool;   // True - prepare data and send a message to the MFC
   END_VAR

   VAR_TEMP
      ts_StringDate : Struct   // Temporary memory with string value
         Year : String;
         Month : String;
         Day : String;
         SorterID : String;
         Code : String;
      END_STRUCT;
      ti_Loop : Int;   // Loop counter
      ti_ObjectID : UDInt;   // Parcel identifier
   END_VAR

   VAR CONSTANT
      ci_MessageLength : Word := 16#0016;   // 10#0021 = 16#0016 - Message length
      ci_Som : Byte := 16#FD;   // Start of message
      ci_Eom : Byte := 16#FE;   // End of message
      ci_MsgID : Word := 16#00C9;   // 10#0201 = 16#00C9 - Message ID
      ci_MsgLength : Word := 16#0012;   // 10#0018 = 16#0012 - Message length
      ci_SourceNode : Int := 1;   // 1 - PLC ID Source Node
      ci_DestinationNode : Int := 2;   // 2 - MFC ID Destination Node
   END_VAR


BEGIN
	(*
	----------------------------------------------------------------------------------------
	|                                                                                      |
	|  Copyright  2023             FORTNA Europe BV                                        |
	|  All Rights Reserved         Netherlands                                             |
	|                                                                                      |
	----------------------------------------------------------------------------------------
	Version history:
	Date        | Version   | Author       | Remark
	----------------------------------------------------------------------------------------
	27/04/2023  | 1.0       | S. Nikodem   | Release TIA 17 | DHL Munich 2023
	13/03/2023  | 1.1       | S. Nieswiec  | Updated for new Baseline
	02/05/2024  | 1.2       | J.Majer      | Datatype conversions changed from automatic to explicit, to accomodate IEC 61131-3 standard

	*)

	REGION 1 – FIFO header status update

	    // Mode 'S' - FIFO register status update.
	    "FC_Fifo"(ic_Mode := 'S',
	              qUDT_Status => #ss_Status.FIFOStatus,
	              qx_Error => #ss_Status.FIFOError,
	              qx_Warning => #ss_Status.FIFOWarning,
	              iqv_Data := #s_UDT_MessageArray,
	              iqUDT_FifoHeader := #iq_UDT_FifoHeader,
	              iqv_DataBuffer := #iqs_FifoData);

	END_REGION

	REGION 2 - Check input data if are if range

	    //Convert 'is_ObjectID' to numeric variable
	    #ti_ObjectID := STRING_TO_UDINT(#is_ObjectID);

	    IF (#ti_ObjectID < 0)
	        OR (#ii_SorterID < 0)
	        OR (#ii_SorterID > 99)
	    THEN
	        #ss_Status.InvalidInputData := True;
	    ELSE
	        #ss_Status.InvalidInputData := FALSE;
	    END_IF;

	END_REGION

	REGION 3 – Data preparation

	    //Send message when is new parcel
	    #sx_NewData := (#is_ObjectID <> #ss_OldObjectID) AND NOT (#is_ObjectID = '0');
	    // Save last value
	    #ss_OldObjectID := #is_ObjectID;

	END_REGION

	REGION 4 – Message array size validation

	    // Get size of the array.
	    #si_MaximumMessageLength := "FC_GetNrOfArrayEl"(#s_UDT_MessageArray.Bytes);

	    // Message array size validation.
	    #ss_Status.InvalidMessageArraySize := WORD_TO_INT(#ci_MessageLength) > #si_MaximumMessageLength;

	END_REGION

	REGION 5 – Message preparation

	    // FIFO full check.
	    IF NOT #iq_UDT_FifoHeader.Status.Full
	    THEN
	        // Errors and send pulse check.
	        IF NOT #ss_Status.FIFOError
	            AND NOT #ss_Status.InvalidMessageArraySize
	            AND NOT #ss_Status.InvalidInputData
	            AND #sx_NewData
	        THEN

	            REGION 5.1 – VID preparation

	                // Convert the year into a character string
	                VAL_STRG(IN := #i_ActualTimeDTL.YEAR,
	                         SIZE := 4,
	                         PREC := 0,
	                         FORMAT := 0,
	                         P := 1,
	                         OUT => #ts_StringDate.Year);

	                // Using the HTA function, convert date into a string format
	                #ss_Status.HTAReturn.Month := HTA(IN := WORD_TO_BYTE(INT_TO_BCD16((USINT_TO_INT(#i_ActualTimeDTL.MONTH)))), N := 1, OUT => #ts_StringDate.Month);   // Convert the month
	                #ss_Status.HTAReturn.Day := HTA(IN := WORD_TO_BYTE(INT_TO_BCD16((USINT_TO_INT(#i_ActualTimeDTL.DAY)))), N := 1, OUT => #ts_StringDate.Day);         // Convert the day

	                //Convert Sorter ID value from number to string
	                #ts_StringDate.SorterID := INT_TO_STRING(#ii_SorterID);

	                //Delete sing '+' from string value
	                IF #ts_StringDate.SorterID[1] = '+' THEN
	                    #ts_StringDate.SorterID := DELETE(IN := #ts_StringDate.SorterID, L := 1, P := 1);
	                END_IF;

	                //Add zero when the variable size is to small
	                IF #ii_SorterID < 10 THEN
	                    #ts_StringDate.SorterID := INSERT(IN1 := #ts_StringDate.SorterID, IN2 := '0', P := 0);
	                END_IF;

	                //Creat ID code - value 000 001 to 999 999
	                #sdi_VIDCode += 1;

	                IF #sdi_VIDCode > 999999 THEN
	                    #sdi_VIDCode := 0;
	                END_IF;

	                //Convert VID code value from number to string
	                #ts_StringDate.Code := DINT_TO_STRING(#sdi_VIDCode);

	                //Delete sing '+' from string
	                IF #ts_StringDate.Code[1] = '+' THEN
	                    #ts_StringDate.Code := DELETE(IN := #ts_StringDate.Code, L := 1, P := 1);
	                END_IF;

	                //Add zero when the variable size is to small
	                IF #sdi_VIDCode < 10 THEN
	                    #ts_StringDate.Code := INSERT(IN1 := #ts_StringDate.Code, IN2 := '00000', P := 0);
	                ELSIF #sdi_VIDCode < 100 THEN
	                    #ts_StringDate.Code := INSERT(IN1 := #ts_StringDate.Code, IN2 := '0000', P := 0);
	                ELSIF #sdi_VIDCode < 1000 THEN
	                    #ts_StringDate.Code := INSERT(IN1 := #ts_StringDate.Code, IN2 := '000', P := 0);
	                ELSIF #sdi_VIDCode < 10000 THEN
	                    #ts_StringDate.Code := INSERT(IN1 := #ts_StringDate.Code, IN2 := '00', P := 0);
	                ELSIF #sdi_VIDCode < 100000 THEN
	                    #ts_StringDate.Code := INSERT(IN1 := #ts_StringDate.Code, IN2 := '0', P := 0);
	                END_IF;

	                //Combine strings
	                #ss_VID := (CONCAT(IN1 := #ts_StringDate.Year,
	                                   IN2 := #ts_StringDate.Month,
	                                   IN3 := #ts_StringDate.Day,
	                                   IN4 := #ts_StringDate.SorterID,
	                                   IN5 := #ts_StringDate.Code));

	                //Convert string value to ASCII
	                FOR #ti_Loop := 1 TO 16 DO
	                    #sa_VIDBytes[#ti_Loop] := CHAR_TO_BYTE(#ss_VID[#ti_Loop]);
	                END_FOR;

	            END_REGION

	            REGION 5.2 – Header preparation

	                // Check sequence number. If it is equal or greater than 255 reset it to 1.
	                IF #iqdi_MessageSequenceNumber <= 255
	                THEN
	                    #iqdi_MessageSequenceNumber += 1;
	                ELSE
	                    #iqdi_MessageSequenceNumber := 1;
	                END_IF;

	                // Write parts of the header into structure.
	                #s_UDT_MessageHeader.SOM := #ci_Som;
	                #s_UDT_MessageHeader.SourceNode := INT_TO_BYTE(#ci_SourceNode);
	                #s_UDT_MessageHeader.DestinationNode := INT_TO_BYTE(#ci_DestinationNode);
	                #s_UDT_MessageHeader.SeqNumber := INT_TO_BYTE(#iqdi_MessageSequenceNumber);
	                #s_UDT_MessageHeader.DataLength := #ci_MessageLength;
	                #s_UDT_MessageHeader.NumMsg := 1;

	                // Write parts of the body into structure.
	                #ss_MessageBody.MsgID := #ci_MsgID;
	                #ss_MessageBody.MsgLength := #ci_MsgLength;
	                #ss_MessageBody.ObjectID := #is_ObjectID;
	                #ss_MessageBody.VID := #sa_VIDBytes;
	                #ss_MessageBody.Eom := #ci_Eom;

	            END_REGION

	            REGION 5.3 – Convert message into array of bytes

	                // Initialize the header serialize position and convert header structure into array of bytes.
	                #sdi_SerializePosition := 0;
	                #si_SerializeStatus := Serialize(SRC_VARIABLE := #s_UDT_MessageHeader,
	                                                 DEST_ARRAY => #s_UDT_MessageArray.Bytes,
	                                                 POS := #sdi_SerializePosition);

	                // Initialize the body serialize position and convert header structure into array of bytes
	                #si_SerializeStatus := Serialize(SRC_VARIABLE := #ss_MessageBody,
	                                                 DEST_ARRAY => #s_UDT_MessageArray.Bytes,
	                                                 POS := #sdi_SerializePosition);

	            END_REGION

	            REGION 5.4 – Write message into the FIFO buffer

	                // Mode 'W' - Write FIFO record.
	                "FC_Fifo"(ic_Mode := 'W',
	                          qUDT_Status => #ss_Status.FIFOStatus,
	                          qx_Error => #ss_Status.FIFOError,
	                          qx_Warning => #ss_Status.FIFOWarning,
	                          iqv_Data := #s_UDT_MessageArray,
	                          iqUDT_FifoHeader := #iq_UDT_FifoHeader,
	                          iqv_DataBuffer := #iqs_FifoData);

	            END_REGION

	        END_IF;
	    ELSE
	        // If FIFO is full set FIFO main and FIFO full errors.
	        #ss_Status.FIFOError := TRUE;
	        #ss_Status.FIFOStatus.FifoFull := TRUE;
	    END_IF;

	END_REGION

	REGION 6 - Status

	    // Parametrization collective error output.
	    #qx_Error :=
	    #ss_Status.FIFOError
	    OR #ss_Status.InvalidTimeInterval
	    OR #ss_Status.InvalidMessageArraySize
	    OR #ss_Status.InvalidInputData;

	    // Parametrization collective warning output.
	    #qx_Warning := #ss_Status.FIFOWarning;

	END_REGION
END_FUNCTION_BLOCK

FUNCTION "FC_EquipmentReport" : Void
TITLE = FC_Equipment_Report
{ S7_Optimized_Access := 'TRUE' }
AUTHOR : MHSE
FAMILY : GeneralSystemFunctions
VERSION : 3.0
// ATTRIBUTES
// AUTO_NUMBER = True
// BLOCK_NUMBER = 16
// END_ATTRIBUTES
//Function to generate equipment report.
   VAR_INPUT
      iUDT_Status : "UDT_CommonStatus";   // Status structure
   END_VAR

   VAR_IN_OUT
      iqUDT_Control : "UDT_EquipmentControl";   // Equipment control
   END_VAR


BEGIN
	(*
	----------------------------------------------------------------------------------------

	Version history:
	Date        | Version   | Author        | Remark
	----------------------------------------------------------------------------------------
	24/05/2019  | 0.1       | F.Baten       | first release MHS TIA 15.1
	17/06/2019  | 0.3       | L.Klar        | Manual mode added to "UDT_EquipmentControl"
	17/07/2019  | 0.4       | A.Nowak       | Add all statuses and comments
	24/07/2019  | 2.0       | L.Klar        | 2.0 MHS library release TIA 15.1
	27/08/2019  | 2.1       | K.Pokorski    | Comments adjusted
	16/09/2019  | 2.2       | K.Pokorski    | Equipment error free condition added to "Restart required" status
	06/10/2019  | 2.3       | S. Deukar     | Updated accoring to new UDT equipment report
	12/11/2019  | 3.0       | P.Majka       | 3.0 MHS library release TIA 15.1
	05/02/2024  | 3.1       | L.Klar        | Auto On extention added
	13/03/2024  | 4.0       | S. Nieswiec   | Added to baseline
	*)

	REGION 1 - Equipment report update

	    // Extension of stopped equipment report with the stopped status
	    #iqUDT_Control.Report.Stopped := #iUDT_Status.Stopped
	    OR #iqUDT_Control.Report.Stopped;

	    // Extension of started equipment report with the started status
	    #iqUDT_Control.Report.Running := #iUDT_Status.Running
	    OR #iqUDT_Control.Report.Running;

	    // Extension of energy save equipment report with the energy save status
	    #iqUDT_Control.Report.EnergySave := #iUDT_Status.EnergySave
	    OR #iqUDT_Control.Report.EnergySave;

	    // Extension of warning equipment report with the warning status
	    #iqUDT_Control.Report.Warning := #iUDT_Status.Warning
	    OR #iqUDT_Control.Report.Warning;

	    // Extension of manual mode equipment report with the manual mode status
	    #iqUDT_Control.Report.Manual := #iUDT_Status.Manual
	    OR #iqUDT_Control.Report.Manual;

	    // Extension of error equipment report with the error status
	    #iqUDT_Control.Report.Error := #iUDT_Status.Error
	    OR #iqUDT_Control.Report.Error;

	    // Extension of safety stop equipment report with the safety stop status
	    #iqUDT_Control.Report.SafetyStop := #iUDT_Status.SafetyStop
	    OR #iqUDT_Control.Report.SafetyStop;

	    // Extension of Auto On equipment report with the Auto On status
	    #iqUDT_Control.Report.AutoON := #iUDT_Status.AutoON
	    OR #iqUDT_Control.Report.AutoON;

	    // Extension of restart required equipment report with the restart required and no equipment error statuses
	    #iqUDT_Control.Request.RestartRequired := #iUDT_Status.Stopped
	    AND NOT #iUDT_Status.Error
	    OR #iqUDT_Control.Request.RestartRequired;

	END_REGION
END_FUNCTION

FUNCTION "FC_TimeDiff" : Void
TITLE = FC_TimeDiff
{ S7_Optimized_Access := 'TRUE' }
AUTHOR : MHSE
FAMILY : GeneralSystemFunctions
VERSION : 3.0
// ATTRIBUTES
// AUTO_NUMBER = True
// BLOCK_NUMBER = 28
// END_ATTRIBUTES
//Function to calculate time difference.
   VAR_INPUT
      is_EarlierTimeAsString : String;   // Earlier time in string
      is_LaterTimeAsString : String;   // Later time in sting
   END_VAR

   VAR_OUTPUT
      qt_TimeDifference : LTime;   // Difference between times
   END_VAR

   VAR_TEMP
      tt_EarlierDate {InstructionName := 'DTL'; LibVersion := '1.0'} : DTL;   // Earlier date in DTL
      tt_LaterDate {InstructionName := 'DTL'; LibVersion := '1.0'} : DTL;   // Later date in DTL
      tt_LaterDateInc {InstructionName := 'DTL'; LibVersion := '1.0'} : DTL;   // Later date in DTL with one additional day
      tt_TimeDifference : LTime;   // Time differance
   END_VAR

   VAR CONSTANT
      ct_OneDay : Time := T#1D;   // One day
   END_VAR


BEGIN
	(*
	----------------------------------------------------------------------------------------

	Version history:
	Date        | Version   | Author        | Remark
	----------------------------------------------------------------------------------------
	24/05/2019  | 0.1       | K.Pokorski    | first release MHS TIA 15.1
	24/07/2019  | 2.0       | L.Klar        | 2.0 MHS library release TIA 15.1
	26/08/2019  | 2.1       | M.Kurpiers    | Comments adjusted
	06/09/2019  | 2.2       | M.Kurpiers    | Change in region 2. Correcting the names of inputs variables.
	21/10/2019  | 2.3       | P.Majka       | Logic changed in region 2 and 3. Simpler checking for the date changed
	12/11/2019  | 3.0       | P.Majka       | 3.0 MHS library release TIA 15.1
	21/02/2023  | 4.0       | F.Baten       | 4.0 Release TIA 17.5
	*)

	REGION 1 - Conversion string TO DTL

	    // Using MHS "FC_StringToTime" standard function convert time in string format to date in DTL format
	    "FC_StringToTime"(is_StringTime := #is_EarlierTimeAsString,
	                      qt_Date => #tt_EarlierDate);

	    "FC_StringToTime"(is_StringTime := #is_LaterTimeAsString,
	                      qt_Date => #tt_LaterDate);

	END_REGION

	REGION 2 - Difference between times

	    // Calculate difference between times
	    #tt_TimeDifference := #tt_LaterDate - #tt_EarlierDate;

	    // Checking the negativity in the time difference
	    IF (LTIME_TO_DINT(#tt_TimeDifference) < 0)
	    THEN

	        // Add one day to later date - later time is smaller than ealier time
	        #tt_LaterDateInc := T_ADD(IN1 := #tt_LaterDate, IN2 := #ct_OneDay);

	        // Calculate difference between times
	        #tt_TimeDifference := #tt_LaterDateInc - #tt_EarlierDate;

	    END_IF;

	END_REGION

	REGION 3 - Write outputs

	    // Saving time difference to the output
	    #qt_TimeDifference := #tt_TimeDifference;

	END_REGION
END_FUNCTION

TYPE "UDT_XrayCommand"
VERSION : 0.1
   STRUCT
      TransportModeOn { ExternalAccessible := 'False'; ExternalVisible := 'False'; ExternalWritable := 'False'} : Bool;   // Command to active the Transport mode
      TransportModeOff { ExternalAccessible := 'False'; ExternalVisible := 'False'; ExternalWritable := 'False'} : Bool;   // Command to deactivate the Transport mode
   END_STRUCT;

END_TYPE

TYPE "UDT_SerialCommunicationReceiveStatus"
VERSION : 0.1
   STRUCT
      NRD : Bool;   // Status from Send_P2P function
      Erro : Bool;   // Status from Send_P2P function
      Status : Word;   // Status from Send_P2P function
      Leng : UInt;   // Status from Send_P2P function
   END_STRUCT;

END_TYPE

TYPE "UDT_ABSwitchStatistics"
TITLE = UDT_VSUStatistics
VERSION : 0.1
//User-defined structure of FB_VerticalSwitch function block statistics.
   STRUCT
      UpTime : "UDT_EventStatistic";   // VSU up time
      DownTime : "UDT_EventStatistic";   // VSU down time
      UpperSwitchArea_Error : "UDT_EventStatistic";   // Error statistics for VSU
      LowerSwitchArea_Error : "UDT_EventStatistic";   // Error statistics for VSU
      UpperEntranceJam_Error : "UDT_EventStatistic";   // Error statistics for VSU
      LowerEntranceJam_Error : "UDT_EventStatistic";   // Error statistics for VSU
   END_STRUCT;

END_TYPE

